KUKA KRL program: kuka-srfPath001.src

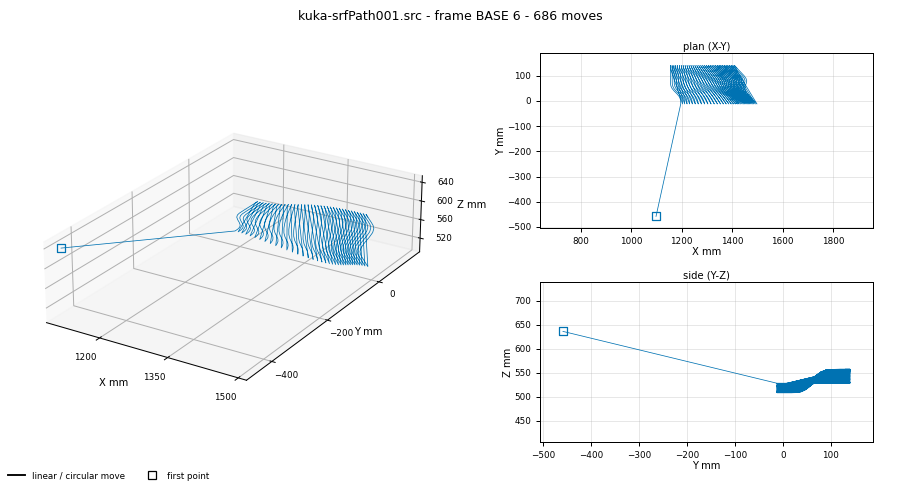
[picture p0: tool path of kuka-srfPath001.src in frame BASE 6, 686 of 688 moves have a stored position in this frame; points joined in program order, loops and branches not executed]
&ACCESS RVP
&REL 1
&PARAM TEMPLATE = C:\KRC\Roboter\Template\vorgabe
&PARAM EDITMASK = *
DEF kuka-srfPath001 ( )
;FOLD INI
;FOLD BASISTECH INI
GLOBAL INTERRUPT DECL 3 WHEN $STOPMESS==TRUE DO IR_STOPM ( )
INTERRUPT ON 3
BAS (#INITMOV,0 )
;ENDFOLD (BASISTECH INI)
;ENDFOLD (INI)
;FOLD STARTPOSITION PTP, VEL 50%, A1 5,A2 -90,A3 100,A4 5,A5 10,A6 -5,E1 0
$BWDSTART = FALSE
PDAT_ACT = {VEL 50,ACC 100,APO_DIST 100}
FDAT_ACT = {TOOL_NO 0,BASE_NO 0,IPO_FRAME #BASE}
BAS (#PTP_PARAMS,50)
$H_POS = {A1 5,A2 -90,A3 100,A4 5,A5 10,A6 -5,E1 0 ,E2 0,E3 0,E4 0,E5 0,E6 0}
PTP  {A1 5,A2 -90,A3 100,A4 5,A5 10,A6 -5,E1 0 ,E2 0,E3 0,E4 0,E5 0,E6 0}
;ENDFOLD
;FOLD SET SPEED TO 50% PTP AND 1 m/sec. LIN
$VEL.CP=1
BAS(#VEL_PTP,50)
BAS(#TOOL,6)
BAS(#BASE,6)
;ENDFOLD
;FOLD PTP FIRST POSITION, VEL= 50 %, TOOL[6], BASE[6]
$BWDSTART = FALSE
PDAT_ACT = {VEL 50,ACC 100,APO_DIST 100}
FDAT_ACT = {TOOL_NO 6,BASE_NO 6,IPO_FRAME #BASE}
BAS (#PTP_PARAMS,50)
;ENDFOLD
PTP {E6POS: X 1098.000, Y -458.000, Z 636.000, A 0.000, B 90.000, C -32.958, E1 0.000, E2 0.0, E3 0.0, E4 0.0, E5 0.0, E6 0.0}
LIN {E6POS: X 1098.000, Y -458.000, Z 636.000, A 0.000, B 90.000, C -32.958, E1 0.000, E2 0.0, E3 0.0, E4 0.0, E5 0.0, E6 0.0} C_DIS
>>>>>>>>>>>>>>>>>>>>>>>>>>>>POWDER FEED ON at=END
>>>>>>>>>>>>>>>>>>>>>>>>>>>>GAS SUPPLY ON at=END
>>>>>>>>>>>>>>>>>>>>>>>>>>>>LASER ON at=END
LIN {E6POS: X 1196.000, Y -12.200, Z 528.000, A 0.000, B 90.000, C -180.000, E1 0.000, E2 0.0, E3 0.0, E4 0.0, E5 0.0, E6 0.0} C_DIS
;POWDER FEED RATE  =  3.0
;LASER INTENSITY  =  4.0
LIN {E6POS: X 1195.747, Y -2.040, Z 528.000, A 90.000, B 90.000, C -90.000, E1 0.000, E2 0.0, E3 0.0, E4 0.0, E5 0.0, E6 0.0} C_DIS
;POWDER FEED RATE  =  3.0
;LASER INTENSITY  =  4.0
LIN {E6POS: X 1193.975, Y 8.120, Z 528.000, A 90.000, B 90.000, C -90.000, E1 0.000, E2 0.0, E3 0.0, E4 0.0, E5 0.0, E6 0.0} C_DIS
;POWDER FEED RATE  =  3.0
;LASER INTENSITY  =  4.0
LIN {E6POS: X 1189.167, Y 18.280, Z 528.000, A -90.000, B 90.000, C 90.000, E1 0.000, E2 0.0, E3 0.0, E4 0.0, E5 0.0, E6 0.0} C_DIS
;POWDER FEED RATE  =  3.0
;LASER INTENSITY  =  4.0
LIN {E6POS: X 1180.562, Y 28.440, Z 528.000, A 90.000, B 90.000, C -90.000, E1 0.000, E2 0.0, E3 0.0, E4 0.0, E5 0.0, E6 0.0} C_DIS
;POWDER FEED RATE  =  3.0
;LASER INTENSITY  =  4.0
LIN {E6POS: X 1170.438, Y 38.600, Z 528.000, A 0.000, B 90.000, C -180.000, E1 0.000, E2 0.0, E3 0.0, E4 0.0, E5 0.0, E6 0.0} C_DIS
;POWDER FEED RATE  =  3.0
;LASER INTENSITY  =  4.0
LIN {E6POS: X 1161.833, Y 48.760, Z 528.000, A 0.000, B 90.000, C -180.000, E1 0.000, E2 0.0, E3 0.0, E4 0.0, E5 0.0, E6 0.0} C_DIS
;POWDER FEED RATE  =  3.0
;LASER INTENSITY  =  4.0
LIN {E6POS: X 1157.025, Y 58.920, Z 528.000, A 0.000, B 90.000, C -180.000, E1 0.000, E2 0.0, E3 0.0, E4 0.0, E5 0.0, E6 0.0} C_DIS
;POWDER FEED RATE  =  3.0
;LASER INTENSITY  =  4.0
LIN {E6POS: X 1155.253, Y 69.080, Z 528.000, A 0.000, B 90.000, C -180.000, E1 0.000, E2 0.0, E3 0.0, E4 0.0, E5 0.0, E6 0.0} C_DIS
;POWDER FEED RATE  =  3.0
;LASER INTENSITY  =  4.0
LIN {E6POS: X 1155.000, Y 79.240, Z 528.000, A 0.000, B 90.000, C -180.000, E1 0.000, E2 0.0, E3 0.0, E4 0.0, E5 0.0, E6 0.0} C_DIS
;POWDER FEED RATE  =  3.0
;LASER INTENSITY  =  4.0
LIN {E6POS: X 1155.000, Y 89.400, Z 528.000, A 0.000, B 90.000, C -180.000, E1 0.000, E2 0.0, E3 0.0, E4 0.0, E5 0.0, E6 0.0} C_DIS
;POWDER FEED RATE  =  3.0
;LASER INTENSITY  =  4.0
LIN {E6POS: X 1155.000, Y 99.560, Z 528.000, A 0.000, B 90.000, C -180.000, E1 0.000, E2 0.0, E3 0.0, E4 0.0, E5 0.0, E6 0.0} C_DIS
;POWDER FEED RATE  =  3.0
;LASER INTENSITY  =  4.0
LIN {E6POS: X 1155.000, Y 109.720, Z 528.000, A 0.000, B 90.000, C -180.000, E1 0.000, E2 0.0, E3 0.0, E4 0.0, E5 0.0, E6 0.0} C_DIS
;POWDER FEED RATE  =  3.0
;LASER INTENSITY  =  4.0
LIN {E6POS: X 1155.000, Y 119.880, Z 528.000, A 0.000, B 90.000, C -180.000, E1 0.000, E2 0.0, E3 0.0, E4 0.0, E5 0.0, E6 0.0} C_DIS
;POWDER FEED RATE  =  3.0
;LASER INTENSITY  =  4.0
LIN {E6POS: X 1155.000, Y 130.040, Z 528.000, A 0.000, B 90.000, C -180.000, E1 0.000, E2 0.0, E3 0.0, E4 0.0, E5 0.0, E6 0.0} C_DIS
;POWDER FEED RATE  =  3.0
;LASER INTENSITY  =  4.0
LIN {E6POS: X 1155.000, Y 140.200, Z 528.000, A 0.000, B 90.000, C -180.000, E1 0.000, E2 0.0, E3 0.0, E4 0.0, E5 0.0, E6 0.0} C_DIS
;POWDER FEED RATE  =  3.0
;LASER INTENSITY  =  4.0
>>>>>>>>>>>>>>>>>>>>>>>>>>>>POWDER FEED OFF  at=START
>>>>>>>>>>>>>>>>>>>>>>>>>>>>LASER OFF at=START
>>>>>>>>>>>>>>>>>>>>>>>>>>>>GAS SUPPLY OFF  at=START
LIN {E6POS: X 1155.000, Y 140.200, Z 528.000, A 0.000, B 90.000, C -180.000, E1 0.000, E2 0.0, E3 0.0, E4 0.0, E5 0.0, E6 0.0} C_DIS
LIN {E6POS: X 1155.000, Y 130.040, Z 528.000, A 0.000, B 90.000, C -180.000, E1 0.000, E2 0.0, E3 0.0, E4 0.0, E5 0.0, E6 0.0} C_DIS
LIN {E6POS: X 1155.000, Y 130.040, Z 528.000, A 0.000, B 90.000, C -180.000, E1 0.000, E2 0.0, E3 0.0, E4 0.0, E5 0.0, E6 0.0} C_DIS
>>>>>>>>>>>>>>>>>>>>>>>>>>>>GAS SUPPLY ON at=END
>>>>>>>>>>>>>>>>>>>>>>>>>>>>POWDER FEED ON at=END
>>>>>>>>>>>>>>>>>>>>>>>>>>>>LASER ON at=END
LIN {E6POS: X 1203.323, Y -12.200, Z 527.825, A -179.740, B 87.512, C 0.260, E1 0.000, E2 0.0, E3 0.0, E4 0.0, E5 0.0, E6 0.0} C_DIS
;POWDER FEED RATE  =  3.0
;LASER INTENSITY  =  4.0
LIN {E6POS: X 1203.025, Y -2.040, Z 527.825, A -175.488, B 87.476, C 4.508, E1 0.000, E2 0.0, E3 0.0, E4 0.0, E5 0.0, E6 0.0} C_DIS
;POWDER FEED RATE  =  3.0
;LASER INTENSITY  =  4.0
LIN {E6POS: X 1201.215, Y 8.120, Z 527.825, A -163.194, B 87.347, C 16.789, E1 0.000, E2 0.0, E3 0.0, E4 0.0, E5 0.0, E6 0.0} C_DIS
;POWDER FEED RATE  =  3.0
;LASER INTENSITY  =  4.0
LIN {E6POS: X 1196.383, Y 18.280, Z 527.825, A -146.024, B 86.920, C 33.938, E1 0.000, E2 0.0, E3 0.0, E4 0.0, E5 0.0, E6 0.0} C_DIS
;POWDER FEED RATE  =  3.0
;LASER INTENSITY  =  4.0
LIN {E6POS: X 1187.773, Y 28.440, Z 527.827, A -136.214, B 86.497, C 43.733, E1 0.000, E2 0.0, E3 0.0, E4 0.0, E5 0.0, E6 0.0} C_DIS
;POWDER FEED RATE  =  3.0
;LASER INTENSITY  =  4.0
LIN {E6POS: X 1177.652, Y 38.600, Z 527.841, A -137.529, B 86.842, C 42.428, E1 0.000, E2 0.0, E3 0.0, E4 0.0, E5 0.0, E6 0.0} C_DIS
;POWDER FEED RATE  =  3.0
;LASER INTENSITY  =  4.0
LIN {E6POS: X 1169.042, Y 48.760, Z 527.878, A -152.965, B 87.985, C 27.020, E1 0.000, E2 0.0, E3 0.0, E4 0.0, E5 0.0, E6 0.0} C_DIS
;POWDER FEED RATE  =  3.0
;LASER INTENSITY  =  4.0
LIN {E6POS: X 1164.211, Y 58.920, Z 527.943, A 168.385, B 89.147, C -11.614, E1 0.000, E2 0.0, E3 0.0, E4 0.0, E5 0.0, E6 0.0} C_DIS
;POWDER FEED RATE  =  3.0
;LASER INTENSITY  =  4.0
LIN {E6POS: X 1162.402, Y 69.080, Z 528.020, A 55.505, B 89.456, C -124.496, E1 0.000, E2 0.0, E3 0.0, E4 0.0, E5 0.0, E6 0.0} C_DIS
;POWDER FEED RATE  =  3.0
;LASER INTENSITY  =  4.0
LIN {E6POS: X 1162.105, Y 79.240, Z 528.086, A 12.952, B 88.664, C -167.052, E1 0.000, E2 0.0, E3 0.0, E4 0.0, E5 0.0, E6 0.0} C_DIS
;POWDER FEED RATE  =  3.0
;LASER INTENSITY  =  4.0
LIN {E6POS: X 1162.059, Y 89.400, Z 528.123, A 4.232, B 88.116, C -175.770, E1 0.000, E2 0.0, E3 0.0, E4 0.0, E5 0.0, E6 0.0} C_DIS
;POWDER FEED RATE  =  3.0
;LASER INTENSITY  =  4.0
LIN {E6POS: X 1162.013, Y 99.560, Z 528.136, A 1.145, B 87.889, C -178.856, E1 0.000, E2 0.0, E3 0.0, E4 0.0, E5 0.0, E6 0.0} C_DIS
;POWDER FEED RATE  =  3.0
;LASER INTENSITY  =  4.0
LIN {E6POS: X 1161.967, Y 109.720, Z 528.138, A 0.260, B 87.832, C -179.740, E1 0.000, E2 0.0, E3 0.0, E4 0.0, E5 0.0, E6 0.0} C_DIS
;POWDER FEED RATE  =  3.0
;LASER INTENSITY  =  4.0
LIN {E6POS: X 1161.921, Y 119.880, Z 528.138, A 0.260, B 87.805, C -179.740, E1 0.000, E2 0.0, E3 0.0, E4 0.0, E5 0.0, E6 0.0} C_DIS
;POWDER FEED RATE  =  3.0
;LASER INTENSITY  =  4.0
LIN {E6POS: X 1161.875, Y 130.040, Z 528.138, A 0.260, B 87.776, C -179.740, E1 0.000, E2 0.0, E3 0.0, E4 0.0, E5 0.0, E6 0.0} C_DIS
;POWDER FEED RATE  =  3.0
;LASER INTENSITY  =  4.0
LIN {E6POS: X 1161.829, Y 140.200, Z 528.138, A 0.260, B 87.747, C -179.740, E1 0.000, E2 0.0, E3 0.0, E4 0.0, E5 0.0, E6 0.0} C_DIS
;POWDER FEED RATE  =  3.0
;LASER INTENSITY  =  4.0
>>>>>>>>>>>>>>>>>>>>>>>>>>>>POWDER FEED OFF  at=START
>>>>>>>>>>>>>>>>>>>>>>>>>>>>LASER OFF at=START
>>>>>>>>>>>>>>>>>>>>>>>>>>>>GAS SUPPLY OFF  at=START
LIN {E6POS: X 1161.829, Y 140.200, Z 528.138, A 0.260, B 87.747, C -179.740, E1 0.000, E2 0.0, E3 0.0, E4 0.0, E5 0.0, E6 0.0} C_DIS
LIN {E6POS: X 1161.875, Y 130.040, Z 528.138, A 0.260, B 87.776, C -179.740, E1 0.000, E2 0.0, E3 0.0, E4 0.0, E5 0.0, E6 0.0} C_DIS
LIN {E6POS: X 1161.875, Y 130.040, Z 528.138, A 0.260, B 87.776, C -179.740, E1 0.000, E2 0.0, E3 0.0, E4 0.0, E5 0.0, E6 0.0} C_DIS
>>>>>>>>>>>>>>>>>>>>>>>>>>>>GAS SUPPLY ON at=END
>>>>>>>>>>>>>>>>>>>>>>>>>>>>POWDER FEED ON at=END
>>>>>>>>>>>>>>>>>>>>>>>>>>>>LASER ON at=END
LIN {E6POS: X 1211.725, Y -12.200, Z 527.328, A -178.991, B 85.857, C 1.007, E1 0.000, E2 0.0, E3 0.0, E4 0.0, E5 0.0, E6 0.0} C_DIS
;POWDER FEED RATE  =  3.0
;LASER INTENSITY  =  4.0
LIN {E6POS: X 1211.298, Y -2.040, Z 527.328, A -174.802, B 85.760, C 5.184, E1 0.000, E2 0.0, E3 0.0, E4 0.0, E5 0.0, E6 0.0} C_DIS
;POWDER FEED RATE  =  3.0
;LASER INTENSITY  =  4.0
LIN {E6POS: X 1209.380, Y 8.120, Z 527.328, A -162.723, B 85.506, C 17.227, E1 0.000, E2 0.0, E3 0.0, E4 0.0, E5 0.0, E6 0.0} C_DIS
;POWDER FEED RATE  =  3.0
;LASER INTENSITY  =  4.0
LIN {E6POS: X 1204.481, Y 18.280, Z 527.328, A -145.872, B 84.767, C 34.017, E1 0.000, E2 0.0, E3 0.0, E4 0.0, E5 0.0, E6 0.0} C_DIS
;POWDER FEED RATE  =  3.0
;LASER INTENSITY  =  4.0
LIN {E6POS: X 1195.856, Y 28.440, Z 527.336, A -136.715, B 84.106, C 43.133, E1 0.000, E2 0.0, E3 0.0, E4 0.0, E5 0.0, E6 0.0} C_DIS
;POWDER FEED RATE  =  3.0
;LASER INTENSITY  =  4.0
LIN {E6POS: X 1185.742, Y 38.600, Z 527.388, A -139.845, B 84.831, C 40.040, E1 0.000, E2 0.0, E3 0.0, E4 0.0, E5 0.0, E6 0.0} C_DIS
;POWDER FEED RATE  =  3.0
;LASER INTENSITY  =  4.0
LIN {E6POS: X 1177.119, Y 48.760, Z 527.530, A -163.042, B 86.819, C 16.934, E1 0.000, E2 0.0, E3 0.0, E4 0.0, E5 0.0, E6 0.0} C_DIS
;POWDER FEED RATE  =  3.0
;LASER INTENSITY  =  4.0
LIN {E6POS: X 1172.225, Y 58.920, Z 527.783, A 139.529, B 88.149, C -40.456, E1 0.000, E2 0.0, E3 0.0, E4 0.0, E5 0.0, E6 0.0} C_DIS
;POWDER FEED RATE  =  3.0
;LASER INTENSITY  =  4.0
LIN {E6POS: X 1170.312, Y 69.080, Z 528.081, A 71.606, B 88.220, C -108.402, E1 0.000, E2 0.0, E3 0.0, E4 0.0, E5 0.0, E6 0.0} C_DIS
;POWDER FEED RATE  =  3.0
;LASER INTENSITY  =  4.0
LIN {E6POS: X 1169.889, Y 79.240, Z 528.334, A 27.036, B 87.418, C -152.987, E1 0.000, E2 0.0, E3 0.0, E4 0.0, E5 0.0, E6 0.0} C_DIS
;POWDER FEED RATE  =  3.0
;LASER INTENSITY  =  4.0
LIN {E6POS: X 1169.712, Y 89.400, Z 528.476, A 9.569, B 86.620, C -170.447, E1 0.000, E2 0.0, E3 0.0, E4 0.0, E5 0.0, E6 0.0} C_DIS
;POWDER FEED RATE  =  3.0
;LASER INTENSITY  =  4.0
LIN {E6POS: X 1169.534, Y 99.560, Z 528.528, A 2.915, B 86.218, C -177.092, E1 0.000, E2 0.0, E3 0.0, E4 0.0, E5 0.0, E6 0.0} C_DIS
;POWDER FEED RATE  =  3.0
;LASER INTENSITY  =  4.0
LIN {E6POS: X 1169.355, Y 109.720, Z 528.536, A 1.009, B 86.082, C -178.993, E1 0.000, E2 0.0, E3 0.0, E4 0.0, E5 0.0, E6 0.0} C_DIS
;POWDER FEED RATE  =  3.0
;LASER INTENSITY  =  4.0
LIN {E6POS: X 1169.176, Y 119.880, Z 528.536, A 1.009, B 85.991, C -178.993, E1 0.000, E2 0.0, E3 0.0, E4 0.0, E5 0.0, E6 0.0} C_DIS
;POWDER FEED RATE  =  3.0
;LASER INTENSITY  =  4.0
LIN {E6POS: X 1168.997, Y 130.040, Z 528.536, A 1.009, B 85.895, C -178.993, E1 0.000, E2 0.0, E3 0.0, E4 0.0, E5 0.0, E6 0.0} C_DIS
;POWDER FEED RATE  =  3.0
;LASER INTENSITY  =  4.0
LIN {E6POS: X 1168.818, Y 140.200, Z 528.536, A 1.009, B 85.794, C -178.993, E1 0.000, E2 0.0, E3 0.0, E4 0.0, E5 0.0, E6 0.0} C_DIS
;POWDER FEED RATE  =  3.0
;LASER INTENSITY  =  4.0
>>>>>>>>>>>>>>>>>>>>>>>>>>>>POWDER FEED OFF  at=START
>>>>>>>>>>>>>>>>>>>>>>>>>>>>LASER OFF at=START
>>>>>>>>>>>>>>>>>>>>>>>>>>>>GAS SUPPLY OFF  at=START
LIN {E6POS: X 1168.818, Y 140.200, Z 528.536, A 1.009, B 85.794, C -178.993, E1 0.000, E2 0.0, E3 0.0, E4 0.0, E5 0.0, E6 0.0} C_DIS
LIN {E6POS: X 1168.997, Y 130.040, Z 528.536, A 1.009, B 85.895, C -178.993, E1 0.000, E2 0.0, E3 0.0, E4 0.0, E5 0.0, E6 0.0} C_DIS
LIN {E6POS: X 1168.997, Y 130.040, Z 528.536, A 1.009, B 85.895, C -178.993, E1 0.000, E2 0.0, E3 0.0, E4 0.0, E5 0.0, E6 0.0} C_DIS
>>>>>>>>>>>>>>>>>>>>>>>>>>>>GAS SUPPLY ON at=END
>>>>>>>>>>>>>>>>>>>>>>>>>>>>POWDER FEED ON at=END
>>>>>>>>>>>>>>>>>>>>>>>>>>>>LASER ON at=END
LIN {E6POS: X 1221.090, Y -12.200, Z 526.549, A -177.798, B 84.710, C 2.192, E1 0.000, E2 0.0, E3 0.0, E4 0.0, E5 0.0, E6 0.0} C_DIS
;POWDER FEED RATE  =  3.0
;LASER INTENSITY  =  4.0
LIN {E6POS: X 1220.457, Y -2.040, Z 526.549, A -173.713, B 84.549, C 6.258, E1 0.000, E2 0.0, E3 0.0, E4 0.0, E5 0.0, E6 0.0} C_DIS
;POWDER FEED RATE  =  3.0
;LASER INTENSITY  =  4.0
LIN {E6POS: X 1218.366, Y 8.120, Z 526.549, A -161.979, B 84.181, C 17.934, E1 0.000, E2 0.0, E3 0.0, E4 0.0, E5 0.0, E6 0.0} C_DIS
;POWDER FEED RATE  =  3.0
;LASER INTENSITY  =  4.0
LIN {E6POS: X 1213.360, Y 18.280, Z 526.549, A -145.631, B 83.214, C 34.181, E1 0.000, E2 0.0, E3 0.0, E4 0.0, E5 0.0, E6 0.0} C_DIS
;POWDER FEED RATE  =  3.0
;LASER INTENSITY  =  4.0
LIN {E6POS: X 1204.712, Y 28.440, Z 526.565, A -137.335, B 82.454, C 42.417, E1 0.000, E2 0.0, E3 0.0, E4 0.0, E5 0.0, E6 0.0} C_DIS
;POWDER FEED RATE  =  3.0
;LASER INTENSITY  =  4.0
LIN {E6POS: X 1194.609, Y 38.600, Z 526.678, A -142.877, B 83.593, C 36.951, E1 0.000, E2 0.0, E3 0.0, E4 0.0, E5 0.0, E6 0.0} C_DIS
;POWDER FEED RATE  =  3.0
;LASER INTENSITY  =  4.0
LIN {E6POS: X 1185.969, Y 48.760, Z 526.986, A -176.728, B 86.064, C 3.265, E1 0.000, E2 0.0, E3 0.0, E4 0.0, E5 0.0, E6 0.0} C_DIS
;POWDER FEED RATE  =  3.0
;LASER INTENSITY  =  4.0
LIN {E6POS: X 1180.978, Y 58.920, Z 527.536, A 121.216, B 86.528, C -58.738, E1 0.000, E2 0.0, E3 0.0, E4 0.0, E5 0.0, E6 0.0} C_DIS
;POWDER FEED RATE  =  3.0
;LASER INTENSITY  =  4.0
LIN {E6POS: X 1178.905, Y 69.080, Z 528.182, A 77.896, B 86.281, C -102.128, E1 0.000, E2 0.0, E3 0.0, E4 0.0, E5 0.0, E6 0.0} C_DIS
;POWDER FEED RATE  =  3.0
;LASER INTENSITY  =  4.0
LIN {E6POS: X 1178.286, Y 79.240, Z 528.732, A 39.861, B 85.985, C -140.208, E1 0.000, E2 0.0, E3 0.0, E4 0.0, E5 0.0, E6 0.0} C_DIS
;POWDER FEED RATE  =  3.0
;LASER INTENSITY  =  4.0
LIN {E6POS: X 1177.904, Y 89.400, Z 529.039, A 15.736, B 85.348, C -164.313, E1 0.000, E2 0.0, E3 0.0, E4 0.0, E5 0.0, E6 0.0} C_DIS
;POWDER FEED RATE  =  3.0
;LASER INTENSITY  =  4.0
LIN {E6POS: X 1177.516, Y 99.560, Z 529.153, A 5.242, B 84.872, C -174.779, E1 0.000, E2 0.0, E3 0.0, E4 0.0, E5 0.0, E6 0.0} C_DIS
;POWDER FEED RATE  =  3.0
;LASER INTENSITY  =  4.0
LIN {E6POS: X 1177.126, Y 109.720, Z 529.169, A 2.202, B 84.658, C -177.808, E1 0.000, E2 0.0, E3 0.0, E4 0.0, E5 0.0, E6 0.0} C_DIS
;POWDER FEED RATE  =  3.0
;LASER INTENSITY  =  4.0
LIN {E6POS: X 1176.735, Y 119.880, Z 529.169, A 2.202, B 84.487, C -177.808, E1 0.000, E2 0.0, E3 0.0, E4 0.0, E5 0.0, E6 0.0} C_DIS
;POWDER FEED RATE  =  3.0
;LASER INTENSITY  =  4.0
LIN {E6POS: X 1176.345, Y 130.040, Z 529.169, A 2.202, B 84.305, C -177.809, E1 0.000, E2 0.0, E3 0.0, E4 0.0, E5 0.0, E6 0.0} C_DIS
;POWDER FEED RATE  =  3.0
;LASER INTENSITY  =  4.0
LIN {E6POS: X 1175.954, Y 140.200, Z 529.169, A 2.202, B 84.110, C -177.810, E1 0.000, E2 0.0, E3 0.0, E4 0.0, E5 0.0, E6 0.0} C_DIS
;POWDER FEED RATE  =  3.0
;LASER INTENSITY  =  4.0
>>>>>>>>>>>>>>>>>>>>>>>>>>>>POWDER FEED OFF  at=START
>>>>>>>>>>>>>>>>>>>>>>>>>>>>LASER OFF at=START
>>>>>>>>>>>>>>>>>>>>>>>>>>>>GAS SUPPLY OFF  at=START
LIN {E6POS: X 1175.954, Y 140.200, Z 529.169, A 2.202, B 84.110, C -177.810, E1 0.000, E2 0.0, E3 0.0, E4 0.0, E5 0.0, E6 0.0} C_DIS
LIN {E6POS: X 1176.345, Y 130.040, Z 529.169, A 2.202, B 84.305, C -177.809, E1 0.000, E2 0.0, E3 0.0, E4 0.0, E5 0.0, E6 0.0} C_DIS
LIN {E6POS: X 1176.345, Y 130.040, Z 529.169, A 2.202, B 84.305, C -177.809, E1 0.000, E2 0.0, E3 0.0, E4 0.0, E5 0.0, E6 0.0} C_DIS
>>>>>>>>>>>>>>>>>>>>>>>>>>>>GAS SUPPLY ON at=END
>>>>>>>>>>>>>>>>>>>>>>>>>>>>POWDER FEED ON at=END
>>>>>>>>>>>>>>>>>>>>>>>>>>>>LASER ON at=END
LIN {E6POS: X 1231.298, Y -12.200, Z 525.527, A -176.212, B 83.899, C 3.767, E1 0.000, E2 0.0, E3 0.0, E4 0.0, E5 0.0, E6 0.0} C_DIS
;POWDER FEED RATE  =  3.0
;LASER INTENSITY  =  4.0
LIN {E6POS: X 1230.390, Y -2.040, Z 525.527, A -172.269, B 83.675, C 7.684, E1 0.000, E2 0.0, E3 0.0, E4 0.0, E5 0.0, E6 0.0} C_DIS
;POWDER FEED RATE  =  3.0
;LASER INTENSITY  =  4.0
LIN {E6POS: X 1228.069, Y 8.120, Z 525.527, A -160.997, B 83.205, C 18.879, E1 0.000, E2 0.0, E3 0.0, E4 0.0, E5 0.0, E6 0.0} C_DIS
;POWDER FEED RATE  =  3.0
;LASER INTENSITY  =  4.0
LIN {E6POS: X 1222.921, Y 18.280, Z 525.527, A -145.313, B 82.075, C 34.430, E1 0.000, E2 0.0, E3 0.0, E4 0.0, E5 0.0, E6 0.0} C_DIS
;POWDER FEED RATE  =  3.0
;LASER INTENSITY  =  4.0
LIN {E6POS: X 1214.242, Y 28.440, Z 525.555, A -138.077, B 81.322, C 41.595, E1 0.000, E2 0.0, E3 0.0, E4 0.0, E5 0.0, E6 0.0} C_DIS
;POWDER FEED RATE  =  3.0
;LASER INTENSITY  =  4.0
LIN {E6POS: X 1204.156, Y 38.600, Z 525.749, A -146.760, B 82.894, C 33.038, E1 0.000, E2 0.0, E3 0.0, E4 0.0, E5 0.0, E6 0.0} C_DIS
;POWDER FEED RATE  =  3.0
;LASER INTENSITY  =  4.0
LIN {E6POS: X 1195.495, Y 48.760, Z 526.275, A 166.884, B 85.317, C -13.074, E1 0.000, E2 0.0, E3 0.0, E4 0.0, E5 0.0, E6 0.0} C_DIS
;POWDER FEED RATE  =  3.0
;LASER INTENSITY  =  4.0
LIN {E6POS: X 1190.382, Y 58.920, Z 527.216, A 110.981, B 84.250, C -68.922, E1 0.000, E2 0.0, E3 0.0, E4 0.0, E5 0.0, E6 0.0} C_DIS
;POWDER FEED RATE  =  3.0
;LASER INTENSITY  =  4.0
LIN {E6POS: X 1188.102, Y 69.080, Z 528.324, A 81.066, B 83.730, C -98.987, E1 0.000, E2 0.0, E3 0.0, E4 0.0, E5 0.0, E6 0.0} C_DIS
;POWDER FEED RATE  =  3.0
;LASER INTENSITY  =  4.0
LIN {E6POS: X 1187.229, Y 79.240, Z 529.265, A 50.146, B 84.221, C -129.997, E1 0.000, E2 0.0, E3 0.0, E4 0.0, E5 0.0, E6 0.0} C_DIS
;POWDER FEED RATE  =  3.0
;LASER INTENSITY  =  4.0
LIN {E6POS: X 1186.576, Y 89.400, Z 529.791, A 22.371, B 84.174, C -157.733, E1 0.000, E2 0.0, E3 0.0, E4 0.0, E5 0.0, E6 0.0} C_DIS
;POWDER FEED RATE  =  3.0
;LASER INTENSITY  =  4.0
LIN {E6POS: X 1185.911, Y 99.560, Z 529.985, A 8.053, B 83.765, C -171.994, E1 0.000, E2 0.0, E3 0.0, E4 0.0, E5 0.0, E6 0.0} C_DIS
;POWDER FEED RATE  =  3.0
;LASER INTENSITY  =  4.0
LIN {E6POS: X 1185.239, Y 109.720, Z 530.013, A 3.788, B 83.492, C -176.236, E1 0.000, E2 0.0, E3 0.0, E4 0.0, E5 0.0, E6 0.0} C_DIS
;POWDER FEED RATE  =  3.0
;LASER INTENSITY  =  4.0
LIN {E6POS: X 1184.566, Y 119.880, Z 530.013, A 3.788, B 83.237, C -176.238, E1 0.000, E2 0.0, E3 0.0, E4 0.0, E5 0.0, E6 0.0} C_DIS
;POWDER FEED RATE  =  3.0
;LASER INTENSITY  =  4.0
LIN {E6POS: X 1183.894, Y 130.040, Z 530.013, A 3.788, B 82.961, C -176.240, E1 0.000, E2 0.0, E3 0.0, E4 0.0, E5 0.0, E6 0.0} C_DIS
;POWDER FEED RATE  =  3.0
;LASER INTENSITY  =  4.0
LIN {E6POS: X 1183.221, Y 140.200, Z 530.013, A 3.788, B 82.662, C -176.243, E1 0.000, E2 0.0, E3 0.0, E4 0.0, E5 0.0, E6 0.0} C_DIS
;POWDER FEED RATE  =  3.0
;LASER INTENSITY  =  4.0
>>>>>>>>>>>>>>>>>>>>>>>>>>>>POWDER FEED OFF  at=START
>>>>>>>>>>>>>>>>>>>>>>>>>>>>LASER OFF at=START
>>>>>>>>>>>>>>>>>>>>>>>>>>>>GAS SUPPLY OFF  at=START
LIN {E6POS: X 1183.221, Y 140.200, Z 530.013, A 3.788, B 82.662, C -176.243, E1 0.000, E2 0.0, E3 0.0, E4 0.0, E5 0.0, E6 0.0} C_DIS
LIN {E6POS: X 1183.894, Y 130.040, Z 530.013, A 3.788, B 82.961, C -176.240, E1 0.000, E2 0.0, E3 0.0, E4 0.0, E5 0.0, E6 0.0} C_DIS
LIN {E6POS: X 1183.894, Y 130.040, Z 530.013, A 3.788, B 82.961, C -176.240, E1 0.000, E2 0.0, E3 0.0, E4 0.0, E5 0.0, E6 0.0} C_DIS
>>>>>>>>>>>>>>>>>>>>>>>>>>>>GAS SUPPLY ON at=END
>>>>>>>>>>>>>>>>>>>>>>>>>>>>POWDER FEED ON at=END
>>>>>>>>>>>>>>>>>>>>>>>>>>>>LASER ON at=END
LIN {E6POS: X 1242.232, Y -12.200, Z 524.303, A -174.283, B 83.319, C 5.679, E1 0.000, E2 0.0, E3 0.0, E4 0.0, E5 0.0, E6 0.0} C_DIS
;POWDER FEED RATE  =  3.0
;LASER INTENSITY  =  4.0
LIN {E6POS: X 1240.988, Y -2.040, Z 524.303, A -170.519, B 83.038, C 9.413, E1 0.000, E2 0.0, E3 0.0, E4 0.0, E5 0.0, E6 0.0} C_DIS
;POWDER FEED RATE  =  3.0
;LASER INTENSITY  =  4.0
LIN {E6POS: X 1238.385, Y 8.120, Z 524.303, A -159.813, B 82.480, C 20.027, E1 0.000, E2 0.0, E3 0.0, E4 0.0, E5 0.0, E6 0.0} C_DIS
;POWDER FEED RATE  =  3.0
;LASER INTENSITY  =  4.0
LIN {E6POS: X 1233.064, Y 18.280, Z 524.303, A -144.927, B 81.238, C 34.757, E1 0.000, E2 0.0, E3 0.0, E4 0.0, E5 0.0, E6 0.0} C_DIS
;POWDER FEED RATE  =  3.0
;LASER INTENSITY  =  4.0
LIN {E6POS: X 1224.347, Y 28.440, Z 524.345, A -138.947, B 80.574, C 40.668, E1 0.000, E2 0.0, E3 0.0, E4 0.0, E5 0.0, E6 0.0} C_DIS
;POWDER FEED RATE  =  3.0
;LASER INTENSITY  =  4.0
LIN {E6POS: X 1214.283, Y 38.600, Z 524.636, A -151.669, B 82.570, C 28.129, E1 0.000, E2 0.0, E3 0.0, E4 0.0, E5 0.0, E6 0.0} C_DIS
;POWDER FEED RATE  =  3.0
;LASER INTENSITY  =  4.0
LIN {E6POS: X 1205.602, Y 48.760, Z 525.427, A 150.464, B 84.256, C -29.412, E1 0.000, E2 0.0, E3 0.0, E4 0.0, E5 0.0, E6 0.0} C_DIS
;POWDER FEED RATE  =  3.0
;LASER INTENSITY  =  4.0
LIN {E6POS: X 1200.350, Y 58.920, Z 526.841, A 104.954, B 81.423, C -74.884, E1 0.000, E2 0.0, E3 0.0, E4 0.0, E5 0.0, E6 0.0} C_DIS
;POWDER FEED RATE  =  3.0
;LASER INTENSITY  =  4.0
LIN {E6POS: X 1197.827, Y 69.080, Z 528.506, A 82.914, B 80.675, C -97.180, E1 0.000, E2 0.0, E3 0.0, E4 0.0, E5 0.0, E6 0.0} C_DIS
;POWDER FEED RATE  =  3.0
;LASER INTENSITY  =  4.0
LIN {E6POS: X 1196.652, Y 79.240, Z 529.920, A 57.886, B 82.098, C -122.360, E1 0.000, E2 0.0, E3 0.0, E4 0.0, E5 0.0, E6 0.0} C_DIS
;POWDER FEED RATE  =  3.0
;LASER INTENSITY  =  4.0
LIN {E6POS: X 1195.673, Y 89.400, Z 530.711, A 29.078, B 83.006, C -151.103, E1 0.000, E2 0.0, E3 0.0, E4 0.0, E5 0.0, E6 0.0} C_DIS
;POWDER FEED RATE  =  3.0
;LASER INTENSITY  =  4.0
LIN {E6POS: X 1194.670, Y 99.560, Z 531.002, A 11.262, B 82.831, C -168.824, E1 0.000, E2 0.0, E3 0.0, E4 0.0, E5 0.0, E6 0.0} C_DIS
;POWDER FEED RATE  =  3.0
;LASER INTENSITY  =  4.0
LIN {E6POS: X 1193.655, Y 109.720, Z 531.044, A 5.717, B 82.530, C -174.331, E1 0.000, E2 0.0, E3 0.0, E4 0.0, E5 0.0, E6 0.0} C_DIS
;POWDER FEED RATE  =  3.0
;LASER INTENSITY  =  4.0
LIN {E6POS: X 1192.638, Y 119.880, Z 531.044, A 5.717, B 82.194, C -174.335, E1 0.000, E2 0.0, E3 0.0, E4 0.0, E5 0.0, E6 0.0} C_DIS
;POWDER FEED RATE  =  3.0
;LASER INTENSITY  =  4.0
LIN {E6POS: X 1191.621, Y 130.040, Z 531.044, A 5.717, B 81.826, C -174.340, E1 0.000, E2 0.0, E3 0.0, E4 0.0, E5 0.0, E6 0.0} C_DIS
;POWDER FEED RATE  =  3.0
;LASER INTENSITY  =  4.0
LIN {E6POS: X 1190.603, Y 140.200, Z 531.044, A 5.717, B 81.422, C -174.346, E1 0.000, E2 0.0, E3 0.0, E4 0.0, E5 0.0, E6 0.0} C_DIS
;POWDER FEED RATE  =  3.0
;LASER INTENSITY  =  4.0
>>>>>>>>>>>>>>>>>>>>>>>>>>>>POWDER FEED OFF  at=START
>>>>>>>>>>>>>>>>>>>>>>>>>>>>LASER OFF at=START
>>>>>>>>>>>>>>>>>>>>>>>>>>>>GAS SUPPLY OFF  at=START
LIN {E6POS: X 1190.603, Y 140.200, Z 531.044, A 5.717, B 81.422, C -174.346, E1 0.000, E2 0.0, E3 0.0, E4 0.0, E5 0.0, E6 0.0} C_DIS
LIN {E6POS: X 1191.621, Y 130.040, Z 531.044, A 5.717, B 81.826, C -174.340, E1 0.000, E2 0.0, E3 0.0, E4 0.0, E5 0.0, E6 0.0} C_DIS
LIN {E6POS: X 1191.621, Y 130.040, Z 531.044, A 5.717, B 81.826, C -174.340, E1 0.000, E2 0.0, E3 0.0, E4 0.0, E5 0.0, E6 0.0} C_DIS
>>>>>>>>>>>>>>>>>>>>>>>>>>>>GAS SUPPLY ON at=END
>>>>>>>>>>>>>>>>>>>>>>>>>>>>POWDER FEED ON at=END
>>>>>>>>>>>>>>>>>>>>>>>>>>>>LASER ON at=END
LIN {E6POS: X 1253.772, Y -12.200, Z 522.917, A -172.066, B 82.909, C 7.874, E1 0.000, E2 0.0, E3 0.0, E4 0.0, E5 0.0, E6 0.0} C_DIS
;POWDER FEED RATE  =  3.0
;LASER INTENSITY  =  4.0
LIN {E6POS: X 1252.140, Y -2.040, Z 522.917, A -168.515, B 82.578, C 11.391, E1 0.000, E2 0.0, E3 0.0, E4 0.0, E5 0.0, E6 0.0} C_DIS
;POWDER FEED RATE  =  3.0
;LASER INTENSITY  =  4.0
LIN {E6POS: X 1249.211, Y 8.120, Z 522.917, A -158.465, B 81.944, C 21.342, E1 0.000, E2 0.0, E3 0.0, E4 0.0, E5 0.0, E6 0.0} C_DIS
;POWDER FEED RATE  =  3.0
;LASER INTENSITY  =  4.0
LIN {E6POS: X 1243.689, Y 18.280, Z 522.917, A -144.486, B 80.635, C 35.152, E1 0.000, E2 0.0, E3 0.0, E4 0.0, E5 0.0, E6 0.0} C_DIS
;POWDER FEED RATE  =  3.0
;LASER INTENSITY  =  4.0
LIN {E6POS: X 1234.929, Y 28.440, Z 522.974, A -139.956, B 80.125, C 39.624, E1 0.000, E2 0.0, E3 0.0, E4 0.0, E5 0.0, E6 0.0} C_DIS
;POWDER FEED RATE  =  3.0
;LASER INTENSITY  =  4.0
LIN {E6POS: X 1224.893, Y 38.600, Z 523.377, A -157.810, B 82.493, C 22.018, E1 0.000, E2 0.0, E3 0.0, E4 0.0, E5 0.0, E6 0.0} C_DIS
;POWDER FEED RATE  =  3.0
;LASER INTENSITY  =  4.0
LIN {E6POS: X 1216.195, Y 48.760, Z 524.470, A 136.592, B 82.733, C -43.178, E1 0.000, E2 0.0, E3 0.0, E4 0.0, E5 0.0, E6 0.0} C_DIS
;POWDER FEED RATE  =  3.0
;LASER INTENSITY  =  4.0
LIN {E6POS: X 1210.792, Y 58.920, Z 526.426, A 101.116, B 78.174, C -78.649, E1 0.000, E2 0.0, E3 0.0, E4 0.0, E5 0.0, E6 0.0} C_DIS
;POWDER FEED RATE  =  3.0
;LASER INTENSITY  =  4.0
LIN {E6POS: X 1208.002, Y 69.080, Z 528.727, A 84.092, B 77.240, C -96.057, E1 0.000, E2 0.0, E3 0.0, E4 0.0, E5 0.0, E6 0.0} C_DIS
;POWDER FEED RATE  =  3.0
;LASER INTENSITY  =  4.0
LIN {E6POS: X 1206.489, Y 79.240, Z 530.684, A 63.606, B 79.659, C -116.769, E1 0.000, E2 0.0, E3 0.0, E4 0.0, E5 0.0, E6 0.0} C_DIS
;POWDER FEED RATE  =  3.0
;LASER INTENSITY  =  4.0
LIN {E6POS: X 1205.139, Y 89.400, Z 531.777, A 35.505, B 81.785, C -144.774, E1 0.000, E2 0.0, E3 0.0, E4 0.0, E5 0.0, E6 0.0} C_DIS
;POWDER FEED RATE  =  3.0
;LASER INTENSITY  =  4.0
LIN {E6POS: X 1203.747, Y 99.560, Z 532.179, A 14.772, B 82.022, C -165.365, E1 0.000, E2 0.0, E3 0.0, E4 0.0, E5 0.0, E6 0.0} C_DIS
;POWDER FEED RATE  =  3.0
;LASER INTENSITY  =  4.0
LIN {E6POS: X 1202.335, Y 109.720, Z 532.237, A 7.934, B 81.732, C -172.148, E1 0.000, E2 0.0, E3 0.0, E4 0.0, E5 0.0, E6 0.0} C_DIS
;POWDER FEED RATE  =  3.0
;LASER INTENSITY  =  4.0
LIN {E6POS: X 1200.919, Y 119.880, Z 532.237, A 7.934, B 81.321, C -172.156, E1 0.000, E2 0.0, E3 0.0, E4 0.0, E5 0.0, E6 0.0} C_DIS
;POWDER FEED RATE  =  3.0
;LASER INTENSITY  =  4.0
LIN {E6POS: X 1199.503, Y 130.040, Z 532.237, A 7.934, B 80.867, C -172.165, E1 0.000, E2 0.0, E3 0.0, E4 0.0, E5 0.0, E6 0.0} C_DIS
;POWDER FEED RATE  =  3.0
;LASER INTENSITY  =  4.0
LIN {E6POS: X 1198.087, Y 140.200, Z 532.237, A 7.934, B 80.363, C -172.177, E1 0.000, E2 0.0, E3 0.0, E4 0.0, E5 0.0, E6 0.0} C_DIS
;POWDER FEED RATE  =  3.0
;LASER INTENSITY  =  4.0
>>>>>>>>>>>>>>>>>>>>>>>>>>>>POWDER FEED OFF  at=START
>>>>>>>>>>>>>>>>>>>>>>>>>>>>LASER OFF at=START
>>>>>>>>>>>>>>>>>>>>>>>>>>>>GAS SUPPLY OFF  at=START
LIN {E6POS: X 1198.087, Y 140.200, Z 532.237, A 7.934, B 80.363, C -172.177, E1 0.000, E2 0.0, E3 0.0, E4 0.0, E5 0.0, E6 0.0} C_DIS
LIN {E6POS: X 1199.503, Y 130.040, Z 532.237, A 7.934, B 80.867, C -172.165, E1 0.000, E2 0.0, E3 0.0, E4 0.0, E5 0.0, E6 0.0} C_DIS
LIN {E6POS: X 1199.503, Y 130.040, Z 532.237, A 7.934, B 80.867, C -172.165, E1 0.000, E2 0.0, E3 0.0, E4 0.0, E5 0.0, E6 0.0} C_DIS
>>>>>>>>>>>>>>>>>>>>>>>>>>>>GAS SUPPLY ON at=END
>>>>>>>>>>>>>>>>>>>>>>>>>>>>POWDER FEED ON at=END
>>>>>>>>>>>>>>>>>>>>>>>>>>>>LASER ON at=END
LIN {E6POS: X 1265.800, Y -12.200, Z 521.408, A -169.621, B 82.629, C 10.295, E1 0.000, E2 0.0, E3 0.0, E4 0.0, E5 0.0, E6 0.0} C_DIS
;POWDER FEED RATE  =  3.0
;LASER INTENSITY  =  4.0
LIN {E6POS: X 1263.735, Y -2.040, Z 521.408, A -166.313, B 82.255, C 13.567, E1 0.000, E2 0.0, E3 0.0, E4 0.0, E5 0.0, E6 0.0} C_DIS
;POWDER FEED RATE  =  3.0
;LASER INTENSITY  =  4.0
LIN {E6POS: X 1260.442, Y 8.120, Z 521.408, A -156.990, B 81.562, C 22.786, E1 0.000, E2 0.0, E3 0.0, E4 0.0, E5 0.0, E6 0.0} C_DIS
;POWDER FEED RATE  =  3.0
;LASER INTENSITY  =  4.0
LIN {E6POS: X 1254.696, Y 18.280, Z 521.408, A -143.998, B 80.222, C 35.604, E1 0.000, E2 0.0, E3 0.0, E4 0.0, E5 0.0, E6 0.0} C_DIS
;POWDER FEED RATE  =  3.0
;LASER INTENSITY  =  4.0
LIN {E6POS: X 1245.888, Y 28.440, Z 521.483, A -141.119, B 79.919, C 38.446, E1 0.000, E2 0.0, E3 0.0, E4 0.0, E5 0.0, E6 0.0} C_DIS
;POWDER FEED RATE  =  3.0
;LASER INTENSITY  =  4.0
LIN {E6POS: X 1235.886, Y 38.600, Z 522.008, A -165.382, B 82.551, C 14.500, E1 0.000, E2 0.0, E3 0.0, E4 0.0, E5 0.0, E6 0.0} C_DIS
;POWDER FEED RATE  =  3.0
;LASER INTENSITY  =  4.0
LIN {E6POS: X 1227.178, Y 48.760, Z 523.435, A 126.019, B 80.769, C -53.625, E1 0.000, E2 0.0, E3 0.0, E4 0.0, E5 0.0, E6 0.0} C_DIS
;POWDER FEED RATE  =  3.0
;LASER INTENSITY  =  4.0
LIN {E6POS: X 1221.620, Y 58.920, Z 525.987, A 98.498, B 74.636, C -81.192, E1 0.000, E2 0.0, E3 0.0, E4 0.0, E5 0.0, E6 0.0} C_DIS
;POWDER FEED RATE  =  3.0
;LASER INTENSITY  =  4.0
LIN {E6POS: X 1218.549, Y 69.080, Z 528.989, A 84.885, B 73.556, C -95.332, E1 0.000, E2 0.0, E3 0.0, E4 0.0, E5 0.0, E6 0.0} C_DIS
;POWDER FEED RATE  =  3.0
;LASER INTENSITY  =  4.0
LIN {E6POS: X 1216.671, Y 79.240, Z 531.541, A 67.857, B 76.982, C -112.669, E1 0.000, E2 0.0, E3 0.0, E4 0.0, E5 0.0, E6 0.0} C_DIS
;POWDER FEED RATE  =  3.0
;LASER INTENSITY  =  4.0
LIN {E6POS: X 1214.916, Y 89.400, Z 532.968, A 41.406, B 80.485, C -138.988, E1 0.000, E2 0.0, E3 0.0, E4 0.0, E5 0.0, E6 0.0} C_DIS
;POWDER FEED RATE  =  3.0
;LASER INTENSITY  =  4.0
LIN {E6POS: X 1213.094, Y 99.560, Z 533.493, A 18.481, B 81.299, C -161.718, E1 0.000, E2 0.0, E3 0.0, E4 0.0, E5 0.0, E6 0.0} C_DIS
;POWDER FEED RATE  =  3.0
;LASER INTENSITY  =  4.0
LIN {E6POS: X 1211.238, Y 109.720, Z 533.568, A 10.379, B 81.066, C -169.745, E1 0.000, E2 0.0, E3 0.0, E4 0.0, E5 0.0, E6 0.0} C_DIS
;POWDER FEED RATE  =  3.0
;LASER INTENSITY  =  4.0
LIN {E6POS: X 1209.378, Y 119.880, Z 533.568, A 10.379, B 80.588, C -169.758, E1 0.000, E2 0.0, E3 0.0, E4 0.0, E5 0.0, E6 0.0} C_DIS
;POWDER FEED RATE  =  3.0
;LASER INTENSITY  =  4.0
LIN {E6POS: X 1207.517, Y 130.040, Z 533.568, A 10.379, B 80.056, C -169.774, E1 0.000, E2 0.0, E3 0.0, E4 0.0, E5 0.0, E6 0.0} C_DIS
;POWDER FEED RATE  =  3.0
;LASER INTENSITY  =  4.0
LIN {E6POS: X 1205.656, Y 140.200, Z 533.568, A 10.379, B 79.461, C -169.793, E1 0.000, E2 0.0, E3 0.0, E4 0.0, E5 0.0, E6 0.0} C_DIS
;POWDER FEED RATE  =  3.0
;LASER INTENSITY  =  4.0
>>>>>>>>>>>>>>>>>>>>>>>>>>>>POWDER FEED OFF  at=START
>>>>>>>>>>>>>>>>>>>>>>>>>>>>LASER OFF at=START
>>>>>>>>>>>>>>>>>>>>>>>>>>>>GAS SUPPLY OFF  at=START
LIN {E6POS: X 1205.656, Y 140.200, Z 533.568, A 10.379, B 79.461, C -169.793, E1 0.000, E2 0.0, E3 0.0, E4 0.0, E5 0.0, E6 0.0} C_DIS
LIN {E6POS: X 1207.517, Y 130.040, Z 533.568, A 10.379, B 80.056, C -169.774, E1 0.000, E2 0.0, E3 0.0, E4 0.0, E5 0.0, E6 0.0} C_DIS
LIN {E6POS: X 1207.517, Y 130.040, Z 533.568, A 10.379, B 80.056, C -169.774, E1 0.000, E2 0.0, E3 0.0, E4 0.0, E5 0.0, E6 0.0} C_DIS
>>>>>>>>>>>>>>>>>>>>>>>>>>>>GAS SUPPLY ON at=END
>>>>>>>>>>>>>>>>>>>>>>>>>>>>POWDER FEED ON at=END
>>>>>>>>>>>>>>>>>>>>>>>>>>>>LASER ON at=END
LIN {E6POS: X 1278.198, Y -12.200, Z 519.817, A -167.011, B 82.455, C 12.881, E1 0.000, E2 0.0, E3 0.0, E4 0.0, E5 0.0, E6 0.0} C_DIS
;POWDER FEED RATE  =  3.0
;LASER INTENSITY  =  4.0
LIN {E6POS: X 1275.663, Y -2.040, Z 519.817, A -163.969, B 82.048, C 15.885, E1 0.000, E2 0.0, E3 0.0, E4 0.0, E5 0.0, E6 0.0} C_DIS
;POWDER FEED RATE  =  3.0
;LASER INTENSITY  =  4.0
LIN {E6POS: X 1271.976, Y 8.120, Z 519.817, A -155.425, B 81.312, C 24.326, E1 0.000, E2 0.0, E3 0.0, E4 0.0, E5 0.0, E6 0.0} C_DIS
;POWDER FEED RATE  =  3.0
;LASER INTENSITY  =  4.0
LIN {E6POS: X 1265.986, Y 18.280, Z 519.817, A -143.476, B 79.977, C 36.103, E1 0.000, E2 0.0, E3 0.0, E4 0.0, E5 0.0, E6 0.0} C_DIS
;POWDER FEED RATE  =  3.0
;LASER INTENSITY  =  4.0
LIN {E6POS: X 1257.127, Y 28.440, Z 519.911, A -142.463, B 79.918, C 37.107, E1 0.000, E2 0.0, E3 0.0, E4 0.0, E5 0.0, E6 0.0} C_DIS
;POWDER FEED RATE  =  3.0
;LASER INTENSITY  =  4.0
LIN {E6POS: X 1247.166, Y 38.600, Z 520.567, A -174.500, B 82.636, C 5.455, E1 0.000, E2 0.0, E3 0.0, E4 0.0, E5 0.0, E6 0.0} C_DIS
;POWDER FEED RATE  =  3.0
;LASER INTENSITY  =  4.0
LIN {E6POS: X 1238.455, Y 48.760, Z 522.350, A 118.231, B 78.461, C -61.279, E1 0.000, E2 0.0, E3 0.0, E4 0.0, E5 0.0, E6 0.0} C_DIS
;POWDER FEED RATE  =  3.0
;LASER INTENSITY  =  4.0
LIN {E6POS: X 1232.746, Y 58.920, Z 525.539, A 96.606, B 70.943, C -83.014, E1 0.000, E2 0.0, E3 0.0, E4 0.0, E5 0.0, E6 0.0} C_DIS
;POWDER FEED RATE  =  3.0
;LASER INTENSITY  =  4.0
LIN {E6POS: X 1229.389, Y 69.080, Z 529.291, A 85.437, B 69.759, C -94.862, E1 0.000, E2 0.0, E3 0.0, E4 0.0, E5 0.0, E6 0.0} C_DIS
;POWDER FEED RATE  =  3.0
;LASER INTENSITY  =  4.0
LIN {E6POS: X 1227.134, Y 79.240, Z 532.480, A 71.063, B 74.152, C -109.629, E1 0.000, E2 0.0, E3 0.0, E4 0.0, E5 0.0, E6 0.0} C_DIS
;POWDER FEED RATE  =  3.0
;LASER INTENSITY  =  4.0
LIN {E6POS: X 1224.948, Y 89.400, Z 534.262, A 46.654, B 79.105, C -133.866, E1 0.000, E2 0.0, E3 0.0, E4 0.0, E5 0.0, E6 0.0} C_DIS
;POWDER FEED RATE  =  3.0
;LASER INTENSITY  =  4.0
LIN {E6POS: X 1222.662, Y 99.560, Z 534.919, A 22.283, B 80.638, C -157.985, E1 0.000, E2 0.0, E3 0.0, E4 0.0, E5 0.0, E6 0.0} C_DIS
;POWDER FEED RATE  =  3.0
;LASER INTENSITY  =  4.0
LIN {E6POS: X 1220.327, Y 109.720, Z 535.013, A 12.989, B 80.508, C -167.183, E1 0.000, E2 0.0, E3 0.0, E4 0.0, E5 0.0, E6 0.0} C_DIS
;POWDER FEED RATE  =  3.0
;LASER INTENSITY  =  4.0
LIN {E6POS: X 1217.983, Y 119.880, Z 535.013, A 12.989, B 79.973, C -167.202, E1 0.000, E2 0.0, E3 0.0, E4 0.0, E5 0.0, E6 0.0} C_DIS
;POWDER FEED RATE  =  3.0
;LASER INTENSITY  =  4.0
LIN {E6POS: X 1215.639, Y 130.040, Z 535.013, A 12.989, B 79.374, C -167.226, E1 0.000, E2 0.0, E3 0.0, E4 0.0, E5 0.0, E6 0.0} C_DIS
;POWDER FEED RATE  =  3.0
;LASER INTENSITY  =  4.0
LIN {E6POS: X 1213.296, Y 140.200, Z 535.013, A 12.989, B 78.699, C -167.254, E1 0.000, E2 0.0, E3 0.0, E4 0.0, E5 0.0, E6 0.0} C_DIS
;POWDER FEED RATE  =  3.0
;LASER INTENSITY  =  4.0
>>>>>>>>>>>>>>>>>>>>>>>>>>>>POWDER FEED OFF  at=START
>>>>>>>>>>>>>>>>>>>>>>>>>>>>LASER OFF at=START
>>>>>>>>>>>>>>>>>>>>>>>>>>>>GAS SUPPLY OFF  at=START
LIN {E6POS: X 1213.296, Y 140.200, Z 535.013, A 12.989, B 78.699, C -167.254, E1 0.000, E2 0.0, E3 0.0, E4 0.0, E5 0.0, E6 0.0} C_DIS
LIN {E6POS: X 1215.639, Y 130.040, Z 535.013, A 12.989, B 79.374, C -167.226, E1 0.000, E2 0.0, E3 0.0, E4 0.0, E5 0.0, E6 0.0} C_DIS
LIN {E6POS: X 1215.639, Y 130.040, Z 535.013, A 12.989, B 79.374, C -167.226, E1 0.000, E2 0.0, E3 0.0, E4 0.0, E5 0.0, E6 0.0} C_DIS
>>>>>>>>>>>>>>>>>>>>>>>>>>>>GAS SUPPLY ON at=END
>>>>>>>>>>>>>>>>>>>>>>>>>>>>POWDER FEED ON at=END
>>>>>>>>>>>>>>>>>>>>>>>>>>>>LASER ON at=END
LIN {E6POS: X 1290.847, Y -12.200, Z 518.184, A -164.298, B 82.376, C 15.570, E1 0.000, E2 0.0, E3 0.0, E4 0.0, E5 0.0, E6 0.0} C_DIS
;POWDER FEED RATE  =  3.0
;LASER INTENSITY  =  4.0
LIN {E6POS: X 1287.813, Y -2.040, Z 518.184, A -161.539, B 81.944, C 18.291, E1 0.000, E2 0.0, E3 0.0, E4 0.0, E5 0.0, E6 0.0} C_DIS
;POWDER FEED RATE  =  3.0
;LASER INTENSITY  =  4.0
LIN {E6POS: X 1283.707, Y 8.120, Z 518.184, A -153.805, B 81.186, C 25.927, E1 0.000, E2 0.0, E3 0.0, E4 0.0, E5 0.0, E6 0.0} C_DIS
;POWDER FEED RATE  =  3.0
;LASER INTENSITY  =  4.0
LIN {E6POS: X 1277.459, Y 18.280, Z 518.184, A -142.929, B 79.887, C 36.640, E1 0.000, E2 0.0, E3 0.0, E4 0.0, E5 0.0, E6 0.0} C_DIS
;POWDER FEED RATE  =  3.0
;LASER INTENSITY  =  4.0
LIN {E6POS: X 1268.546, Y 28.440, Z 518.297, A -144.023, B 80.098, C 35.569, E1 0.000, E2 0.0, E3 0.0, E4 0.0, E5 0.0, E6 0.0} C_DIS
;POWDER FEED RATE  =  3.0
;LASER INTENSITY  =  4.0
LIN {E6POS: X 1258.632, Y 38.600, Z 519.090, A 174.940, B 82.643, C -5.019, E1 0.000, E2 0.0, E3 0.0, E4 0.0, E5 0.0, E6 0.0} C_DIS
;POWDER FEED RATE  =  3.0
;LASER INTENSITY  =  4.0
LIN {E6POS: X 1249.930, Y 48.760, Z 521.244, A 112.451, B 75.917, C -66.925, E1 0.000, E2 0.0, E3 0.0, E4 0.0, E5 0.0, E6 0.0} C_DIS
;POWDER FEED RATE  =  3.0
;LASER INTENSITY  =  4.0
LIN {E6POS: X 1244.082, Y 58.920, Z 525.098, A 95.170, B 67.222, C -84.396, E1 0.000, E2 0.0, E3 0.0, E4 0.0, E5 0.0, E6 0.0} C_DIS
;POWDER FEED RATE  =  3.0
;LASER INTENSITY  =  4.0
LIN {E6POS: X 1240.446, Y 69.080, Z 529.632, A 85.827, B 65.979, C -94.567, E1 0.000, E2 0.0, E3 0.0, E4 0.0, E5 0.0, E6 0.0} C_DIS
;POWDER FEED RATE  =  3.0
;LASER INTENSITY  =  4.0
LIN {E6POS: X 1237.811, Y 79.240, Z 533.486, A 73.523, B 71.263, C -107.345, E1 0.000, E2 0.0, E3 0.0, E4 0.0, E5 0.0, E6 0.0} C_DIS
;POWDER FEED RATE  =  3.0
;LASER INTENSITY  =  4.0
LIN {E6POS: X 1235.178, Y 89.400, Z 535.640, A 51.226, B 77.665, C -129.429, E1 0.000, E2 0.0, E3 0.0, E4 0.0, E5 0.0, E6 0.0} C_DIS
;POWDER FEED RATE  =  3.0
;LASER INTENSITY  =  4.0
LIN {E6POS: X 1232.404, Y 99.560, Z 536.433, A 26.080, B 80.022, C -154.263, E1 0.000, E2 0.0, E3 0.0, E4 0.0, E5 0.0, E6 0.0} C_DIS
;POWDER FEED RATE  =  3.0
;LASER INTENSITY  =  4.0
LIN {E6POS: X 1229.560, Y 109.720, Z 536.547, A 15.702, B 80.042, C -164.523, E1 0.000, E2 0.0, E3 0.0, E4 0.0, E5 0.0, E6 0.0} C_DIS
;POWDER FEED RATE  =  3.0
;LASER INTENSITY  =  4.0
LIN {E6POS: X 1226.703, Y 119.880, Z 536.547, A 15.702, B 79.459, C -164.550, E1 0.000, E2 0.0, E3 0.0, E4 0.0, E5 0.0, E6 0.0} C_DIS
;POWDER FEED RATE  =  3.0
;LASER INTENSITY  =  4.0
LIN {E6POS: X 1223.847, Y 130.040, Z 536.547, A 15.702, B 78.804, C -164.582, E1 0.000, E2 0.0, E3 0.0, E4 0.0, E5 0.0, E6 0.0} C_DIS
;POWDER FEED RATE  =  3.0
;LASER INTENSITY  =  4.0
LIN {E6POS: X 1220.991, Y 140.200, Z 536.547, A 15.702, B 78.064, C -164.621, E1 0.000, E2 0.0, E3 0.0, E4 0.0, E5 0.0, E6 0.0} C_DIS
;POWDER FEED RATE  =  3.0
;LASER INTENSITY  =  4.0
>>>>>>>>>>>>>>>>>>>>>>>>>>>>POWDER FEED OFF  at=START
>>>>>>>>>>>>>>>>>>>>>>>>>>>>LASER OFF at=START
>>>>>>>>>>>>>>>>>>>>>>>>>>>>GAS SUPPLY OFF  at=START
LIN {E6POS: X 1220.991, Y 140.200, Z 536.547, A 15.702, B 78.064, C -164.621, E1 0.000, E2 0.0, E3 0.0, E4 0.0, E5 0.0, E6 0.0} C_DIS
LIN {E6POS: X 1223.847, Y 130.040, Z 536.547, A 15.702, B 78.804, C -164.582, E1 0.000, E2 0.0, E3 0.0, E4 0.0, E5 0.0, E6 0.0} C_DIS
LIN {E6POS: X 1223.847, Y 130.040, Z 536.547, A 15.702, B 78.804, C -164.582, E1 0.000, E2 0.0, E3 0.0, E4 0.0, E5 0.0, E6 0.0} C_DIS
>>>>>>>>>>>>>>>>>>>>>>>>>>>>GAS SUPPLY ON at=END
>>>>>>>>>>>>>>>>>>>>>>>>>>>>POWDER FEED ON at=END
>>>>>>>>>>>>>>>>>>>>>>>>>>>>LASER ON at=END
LIN {E6POS: X 1303.630, Y -12.200, Z 516.548, A -161.545, B 82.390, C 18.304, E1 0.000, E2 0.0, E3 0.0, E4 0.0, E5 0.0, E6 0.0} C_DIS
;POWDER FEED RATE  =  3.0
;LASER INTENSITY  =  4.0
LIN {E6POS: X 1300.075, Y -2.040, Z 516.548, A -159.077, B 81.945, C 20.734, E1 0.000, E2 0.0, E3 0.0, E4 0.0, E5 0.0, E6 0.0} C_DIS
;POWDER FEED RATE  =  3.0
;LASER INTENSITY  =  4.0
LIN {E6POS: X 1295.532, Y 8.120, Z 516.548, A -152.163, B 81.185, C 27.557, E1 0.000, E2 0.0, E3 0.0, E4 0.0, E5 0.0, E6 0.0} C_DIS
;POWDER FEED RATE  =  3.0
;LASER INTENSITY  =  4.0
LIN {E6POS: X 1289.015, Y 18.280, Z 516.548, A -142.368, B 79.949, C 37.204, E1 0.000, E2 0.0, E3 0.0, E4 0.0, E5 0.0, E6 0.0} C_DIS
;POWDER FEED RATE  =  3.0
;LASER INTENSITY  =  4.0
LIN {E6POS: X 1280.046, Y 28.440, Z 516.681, A -145.862, B 80.446, C 33.767, E1 0.000, E2 0.0, E3 0.0, E4 0.0, E5 0.0, E6 0.0} C_DIS
;POWDER FEED RATE  =  3.0
;LASER INTENSITY  =  4.0
LIN {E6POS: X 1270.187, Y 38.600, Z 517.615, A 163.374, B 82.480, C -16.491, E1 0.000, E2 0.0, E3 0.0, E4 0.0, E5 0.0, E6 0.0} C_DIS
;POWDER FEED RATE  =  3.0
;LASER INTENSITY  =  4.0
LIN {E6POS: X 1261.508, Y 48.760, Z 520.148, A 108.050, B 73.239, C -71.204, E1 0.000, E2 0.0, E3 0.0, E4 0.0, E5 0.0, E6 0.0} C_DIS
;POWDER FEED RATE  =  3.0
;LASER INTENSITY  =  4.0
LIN {E6POS: X 1255.539, Y 58.920, Z 524.681, A 94.028, B 63.586, C -85.505, E1 0.000, E2 0.0, E3 0.0, E4 0.0, E5 0.0, E6 0.0} C_DIS
;POWDER FEED RATE  =  3.0
;LASER INTENSITY  =  4.0
LIN {E6POS: X 1251.642, Y 69.080, Z 530.013, A 86.100, B 62.328, C -94.401, E1 0.000, E2 0.0, E3 0.0, E4 0.0, E5 0.0, E6 0.0} C_DIS
;POWDER FEED RATE  =  3.0
;LASER INTENSITY  =  4.0
LIN {E6POS: X 1248.635, Y 79.240, Z 534.546, A 75.444, B 68.399, C -105.604, E1 0.000, E2 0.0, E3 0.0, E4 0.0, E5 0.0, E6 0.0} C_DIS
;POWDER FEED RATE  =  3.0
;LASER INTENSITY  =  4.0
LIN {E6POS: X 1245.550, Y 89.400, Z 537.079, A 55.160, B 76.198, C -125.631, E1 0.000, E2 0.0, E3 0.0, E4 0.0, E5 0.0, E6 0.0} C_DIS
;POWDER FEED RATE  =  3.0
;LASER INTENSITY  =  4.0
LIN {E6POS: X 1242.273, Y 99.560, Z 538.012, A 29.788, B 79.446, C -150.632, E1 0.000, E2 0.0, E3 0.0, E4 0.0, E5 0.0, E6 0.0} C_DIS
;POWDER FEED RATE  =  3.0
;LASER INTENSITY  =  4.0
LIN {E6POS: X 1238.898, Y 109.720, Z 538.146, A 18.455, B 79.658, C -161.825, E1 0.000, E2 0.0, E3 0.0, E4 0.0, E5 0.0, E6 0.0} C_DIS
;POWDER FEED RATE  =  3.0
;LASER INTENSITY  =  4.0
LIN {E6POS: X 1235.507, Y 119.880, Z 538.146, A 18.455, B 79.038, C -161.859, E1 0.000, E2 0.0, E3 0.0, E4 0.0, E5 0.0, E6 0.0} C_DIS
;POWDER FEED RATE  =  3.0
;LASER INTENSITY  =  4.0
LIN {E6POS: X 1232.117, Y 130.040, Z 538.146, A 18.455, B 78.340, C -161.900, E1 0.000, E2 0.0, E3 0.0, E4 0.0, E5 0.0, E6 0.0} C_DIS
;POWDER FEED RATE  =  3.0
;LASER INTENSITY  =  4.0
LIN {E6POS: X 1228.726, Y 140.200, Z 538.146, A 18.455, B 77.549, C -161.950, E1 0.000, E2 0.0, E3 0.0, E4 0.0, E5 0.0, E6 0.0} C_DIS
;POWDER FEED RATE  =  3.0
;LASER INTENSITY  =  4.0
>>>>>>>>>>>>>>>>>>>>>>>>>>>>POWDER FEED OFF  at=START
>>>>>>>>>>>>>>>>>>>>>>>>>>>>LASER OFF at=START
>>>>>>>>>>>>>>>>>>>>>>>>>>>>GAS SUPPLY OFF  at=START
LIN {E6POS: X 1228.726, Y 140.200, Z 538.146, A 18.455, B 77.549, C -161.950, E1 0.000, E2 0.0, E3 0.0, E4 0.0, E5 0.0, E6 0.0} C_DIS
LIN {E6POS: X 1232.117, Y 130.040, Z 538.146, A 18.455, B 78.340, C -161.900, E1 0.000, E2 0.0, E3 0.0, E4 0.0, E5 0.0, E6 0.0} C_DIS
LIN {E6POS: X 1232.117, Y 130.040, Z 538.146, A 18.455, B 78.340, C -161.900, E1 0.000, E2 0.0, E3 0.0, E4 0.0, E5 0.0, E6 0.0} C_DIS
>>>>>>>>>>>>>>>>>>>>>>>>>>>>GAS SUPPLY ON at=END
>>>>>>>>>>>>>>>>>>>>>>>>>>>>POWDER FEED ON at=END
>>>>>>>>>>>>>>>>>>>>>>>>>>>>LASER ON at=END
LIN {E6POS: X 1316.427, Y -12.200, Z 514.950, A -158.811, B 82.506, C 21.024, E1 0.000, E2 0.0, E3 0.0, E4 0.0, E5 0.0, E6 0.0} C_DIS
;POWDER FEED RATE  =  3.0
;LASER INTENSITY  =  4.0
LIN {E6POS: X 1312.338, Y -2.040, Z 514.950, A -156.635, B 82.060, C 23.165, E1 0.000, E2 0.0, E3 0.0, E4 0.0, E5 0.0, E6 0.0} C_DIS
;POWDER FEED RATE  =  3.0
;LASER INTENSITY  =  4.0
LIN {E6POS: X 1307.348, Y 8.120, Z 514.950, A -150.529, B 81.318, C 29.189, E1 0.000, E2 0.0, E3 0.0, E4 0.0, E5 0.0, E6 0.0} C_DIS
;POWDER FEED RATE  =  3.0
;LASER INTENSITY  =  4.0
LIN {E6POS: X 1300.555, Y 18.280, Z 514.950, A -141.801, B 80.171, C 37.788, E1 0.000, E2 0.0, E3 0.0, E4 0.0, E5 0.0, E6 0.0} C_DIS
;POWDER FEED RATE  =  3.0
;LASER INTENSITY  =  4.0
LIN {E6POS: X 1291.529, Y 28.440, Z 515.104, A -148.080, B 80.957, C 31.599, E1 0.000, E2 0.0, E3 0.0, E4 0.0, E5 0.0, E6 0.0} C_DIS
;POWDER FEED RATE  =  3.0
;LASER INTENSITY  =  4.0
LIN {E6POS: X 1281.732, Y 38.600, Z 516.177, A 151.531, B 82.084, C -28.239, E1 0.000, E2 0.0, E3 0.0, E4 0.0, E5 0.0, E6 0.0} C_DIS
;POWDER FEED RATE  =  3.0
;LASER INTENSITY  =  4.0
LIN {E6POS: X 1273.093, Y 48.760, Z 519.090, A 104.581, B 70.517, C -74.574, E1 0.000, E2 0.0, E3 0.0, E4 0.0, E5 0.0, E6 0.0} C_DIS
;POWDER FEED RATE  =  3.0
;LASER INTENSITY  =  4.0
LIN {E6POS: X 1267.029, Y 58.920, Z 524.302, A 93.079, B 60.127, C -86.451, E1 0.000, E2 0.0, E3 0.0, E4 0.0, E5 0.0, E6 0.0} C_DIS
;POWDER FEED RATE  =  3.0
;LASER INTENSITY  =  4.0
LIN {E6POS: X 1262.898, Y 69.080, Z 530.434, A 86.285, B 58.893, C -94.337, E1 0.000, E2 0.0, E3 0.0, E4 0.0, E5 0.0, E6 0.0} C_DIS
;POWDER FEED RATE  =  3.0
;LASER INTENSITY  =  4.0
LIN {E6POS: X 1259.539, Y 79.240, Z 535.646, A 76.965, B 65.637, C -104.259, E1 0.000, E2 0.0, E3 0.0, E4 0.0, E5 0.0, E6 0.0} C_DIS
;POWDER FEED RATE  =  3.0
;LASER INTENSITY  =  4.0
LIN {E6POS: X 1256.008, Y 89.400, Z 538.559, A 58.527, B 74.741, C -122.396, E1 0.000, E2 0.0, E3 0.0, E4 0.0, E5 0.0, E6 0.0} C_DIS
;POWDER FEED RATE  =  3.0
;LASER INTENSITY  =  4.0
LIN {E6POS: X 1252.219, Y 99.560, Z 539.632, A 33.340, B 78.915, C -147.153, E1 0.000, E2 0.0, E3 0.0, E4 0.0, E5 0.0, E6 0.0} C_DIS
;POWDER FEED RATE  =  3.0
;LASER INTENSITY  =  4.0
LIN {E6POS: X 1248.302, Y 109.720, Z 539.785, A 21.189, B 79.354, C -159.144, E1 0.000, E2 0.0, E3 0.0, E4 0.0, E5 0.0, E6 0.0} C_DIS
;POWDER FEED RATE  =  3.0
;LASER INTENSITY  =  4.0
LIN {E6POS: X 1244.364, Y 119.880, Z 539.785, A 21.189, B 78.708, C -159.185, E1 0.000, E2 0.0, E3 0.0, E4 0.0, E5 0.0, E6 0.0} C_DIS
;POWDER FEED RATE  =  3.0
;LASER INTENSITY  =  4.0
LIN {E6POS: X 1240.425, Y 130.040, Z 539.785, A 21.189, B 77.980, C -159.235, E1 0.000, E2 0.0, E3 0.0, E4 0.0, E5 0.0, E6 0.0} C_DIS
;POWDER FEED RATE  =  3.0
;LASER INTENSITY  =  4.0
LIN {E6POS: X 1236.486, Y 140.200, Z 539.785, A 21.189, B 77.153, C -159.296, E1 0.000, E2 0.0, E3 0.0, E4 0.0, E5 0.0, E6 0.0} C_DIS
;POWDER FEED RATE  =  3.0
;LASER INTENSITY  =  4.0
>>>>>>>>>>>>>>>>>>>>>>>>>>>>POWDER FEED OFF  at=START
>>>>>>>>>>>>>>>>>>>>>>>>>>>>LASER OFF at=START
>>>>>>>>>>>>>>>>>>>>>>>>>>>>GAS SUPPLY OFF  at=START
LIN {E6POS: X 1236.486, Y 140.200, Z 539.785, A 21.189, B 77.153, C -159.296, E1 0.000, E2 0.0, E3 0.0, E4 0.0, E5 0.0, E6 0.0} C_DIS
LIN {E6POS: X 1240.425, Y 130.040, Z 539.785, A 21.189, B 77.980, C -159.235, E1 0.000, E2 0.0, E3 0.0, E4 0.0, E5 0.0, E6 0.0} C_DIS
LIN {E6POS: X 1240.425, Y 130.040, Z 539.785, A 21.189, B 77.980, C -159.235, E1 0.000, E2 0.0, E3 0.0, E4 0.0, E5 0.0, E6 0.0} C_DIS
>>>>>>>>>>>>>>>>>>>>>>>>>>>>GAS SUPPLY ON at=END
>>>>>>>>>>>>>>>>>>>>>>>>>>>>POWDER FEED ON at=END
>>>>>>>>>>>>>>>>>>>>>>>>>>>>LASER ON at=END
LIN {E6POS: X 1329.120, Y -12.200, Z 513.430, A -156.149, B 82.743, C 23.681, E1 0.000, E2 0.0, E3 0.0, E4 0.0, E5 0.0, E6 0.0} C_DIS
;POWDER FEED RATE  =  3.0
;LASER INTENSITY  =  4.0
LIN {E6POS: X 1324.492, Y -2.040, Z 513.430, A -154.256, B 82.307, C 25.542, E1 0.000, E2 0.0, E3 0.0, E4 0.0, E5 0.0, E6 0.0} C_DIS
;POWDER FEED RATE  =  3.0
;LASER INTENSITY  =  4.0
LIN {E6POS: X 1319.049, Y 8.120, Z 513.430, A -148.931, B 81.605, C 30.797, E1 0.000, E2 0.0, E3 0.0, E4 0.0, E5 0.0, E6 0.0} C_DIS
;POWDER FEED RATE  =  3.0
;LASER INTENSITY  =  4.0
LIN {E6POS: X 1311.978, Y 18.280, Z 513.430, A -141.237, B 80.569, C 38.383, E1 0.000, E2 0.0, E3 0.0, E4 0.0, E5 0.0, E6 0.0} C_DIS
;POWDER FEED RATE  =  3.0
;LASER INTENSITY  =  4.0
LIN {E6POS: X 1302.897, Y 28.440, Z 513.603, A -150.854, B 81.634, C 28.885, E1 0.000, E2 0.0, E3 0.0, E4 0.0, E5 0.0, E6 0.0} C_DIS
;POWDER FEED RATE  =  3.0
;LASER INTENSITY  =  4.0
LIN {E6POS: X 1293.168, Y 38.600, Z 514.814, A 140.163, B 81.430, C -39.521, E1 0.000, E2 0.0, E3 0.0, E4 0.0, E5 0.0, E6 0.0} C_DIS
;POWDER FEED RATE  =  3.0
;LASER INTENSITY  =  4.0
LIN {E6POS: X 1284.589, Y 48.760, Z 518.099, A 101.741, B 67.826, C -77.351, E1 0.000, E2 0.0, E3 0.0, E4 0.0, E5 0.0, E6 0.0} C_DIS
;POWDER FEED RATE  =  3.0
;LASER INTENSITY  =  4.0
LIN {E6POS: X 1278.465, Y 58.920, Z 523.978, A 92.254, B 56.915, C -87.310, E1 0.000, E2 0.0, E3 0.0, E4 0.0, E5 0.0, E6 0.0} C_DIS
;POWDER FEED RATE  =  3.0
;LASER INTENSITY  =  4.0
LIN {E6POS: X 1274.137, Y 69.080, Z 530.894, A 86.397, B 55.740, C -94.357, E1 0.000, E2 0.0, E3 0.0, E4 0.0, E5 0.0, E6 0.0} C_DIS
;POWDER FEED RATE  =  3.0
;LASER INTENSITY  =  4.0
LIN {E6POS: X 1270.457, Y 79.240, Z 536.773, A 78.187, B 63.043, C -103.206, E1 0.000, E2 0.0, E3 0.0, E4 0.0, E5 0.0, E6 0.0} C_DIS
;POWDER FEED RATE  =  3.0
;LASER INTENSITY  =  4.0
LIN {E6POS: X 1266.494, Y 89.400, Z 540.058, A 61.409, B 73.335, C -119.636, E1 0.000, E2 0.0, E3 0.0, E4 0.0, E5 0.0, E6 0.0} C_DIS
;POWDER FEED RATE  =  3.0
;LASER INTENSITY  =  4.0
LIN {E6POS: X 1262.197, Y 99.560, Z 541.268, A 36.692, B 78.439, C -143.869, E1 0.000, E2 0.0, E3 0.0, E4 0.0, E5 0.0, E6 0.0} C_DIS
;POWDER FEED RATE  =  3.0
;LASER INTENSITY  =  4.0
LIN {E6POS: X 1257.733, Y 109.720, Z 541.441, A 23.851, B 79.133, C -156.530, E1 0.000, E2 0.0, E3 0.0, E4 0.0, E5 0.0, E6 0.0} C_DIS
;POWDER FEED RATE  =  3.0
;LASER INTENSITY  =  4.0
LIN {E6POS: X 1253.241, Y 119.880, Z 541.441, A 23.851, B 78.473, C -156.577, E1 0.000, E2 0.0, E3 0.0, E4 0.0, E5 0.0, E6 0.0} C_DIS
;POWDER FEED RATE  =  3.0
;LASER INTENSITY  =  4.0
LIN {E6POS: X 1248.749, Y 130.040, Z 541.441, A 23.851, B 77.730, C -156.635, E1 0.000, E2 0.0, E3 0.0, E4 0.0, E5 0.0, E6 0.0} C_DIS
;POWDER FEED RATE  =  3.0
;LASER INTENSITY  =  4.0
LIN {E6POS: X 1244.257, Y 140.200, Z 541.441, A 23.851, B 76.885, C -156.704, E1 0.000, E2 0.0, E3 0.0, E4 0.0, E5 0.0, E6 0.0} C_DIS
;POWDER FEED RATE  =  3.0
;LASER INTENSITY  =  4.0
>>>>>>>>>>>>>>>>>>>>>>>>>>>>POWDER FEED OFF  at=START
>>>>>>>>>>>>>>>>>>>>>>>>>>>>LASER OFF at=START
>>>>>>>>>>>>>>>>>>>>>>>>>>>>GAS SUPPLY OFF  at=START
LIN {E6POS: X 1244.257, Y 140.200, Z 541.441, A 23.851, B 76.885, C -156.704, E1 0.000, E2 0.0, E3 0.0, E4 0.0, E5 0.0, E6 0.0} C_DIS
LIN {E6POS: X 1248.749, Y 130.040, Z 541.441, A 23.851, B 77.730, C -156.635, E1 0.000, E2 0.0, E3 0.0, E4 0.0, E5 0.0, E6 0.0} C_DIS
LIN {E6POS: X 1248.749, Y 130.040, Z 541.441, A 23.851, B 77.730, C -156.635, E1 0.000, E2 0.0, E3 0.0, E4 0.0, E5 0.0, E6 0.0} C_DIS
>>>>>>>>>>>>>>>>>>>>>>>>>>>>GAS SUPPLY ON at=END
>>>>>>>>>>>>>>>>>>>>>>>>>>>>POWDER FEED ON at=END
>>>>>>>>>>>>>>>>>>>>>>>>>>>>LASER ON at=END
LIN {E6POS: X 1341.590, Y -12.200, Z 512.028, A -153.604, B 83.129, C 26.232, E1 0.000, E2 0.0, E3 0.0, E4 0.0, E5 0.0, E6 0.0} C_DIS
;POWDER FEED RATE  =  3.0
;LASER INTENSITY  =  4.0
LIN {E6POS: X 1336.426, Y -2.040, Z 512.028, A -151.980, B 82.717, C 27.828, E1 0.000, E2 0.0, E3 0.0, E4 0.0, E5 0.0, E6 0.0} C_DIS
;POWDER FEED RATE  =  3.0
;LASER INTENSITY  =  4.0
LIN {E6POS: X 1330.534, Y 8.120, Z 512.028, A -147.392, B 82.075, C 32.358, E1 0.000, E2 0.0, E3 0.0, E4 0.0, E5 0.0, E6 0.0} C_DIS
;POWDER FEED RATE  =  3.0
;LASER INTENSITY  =  4.0
LIN {E6POS: X 1323.184, Y 18.280, Z 512.028, A -140.684, B 81.170, C 38.981, E1 0.000, E2 0.0, E3 0.0, E4 0.0, E5 0.0, E6 0.0} C_DIS
;POWDER FEED RATE  =  3.0
;LASER INTENSITY  =  4.0
LIN {E6POS: X 1314.050, Y 28.440, Z 512.220, A -154.521, B 82.484, C 25.288, E1 0.000, E2 0.0, E3 0.0, E4 0.0, E5 0.0, E6 0.0} C_DIS
;POWDER FEED RATE  =  3.0
;LASER INTENSITY  =  4.0
LIN {E6POS: X 1304.399, Y 38.600, Z 513.562, A 129.749, B 80.529, C -49.864, E1 0.000, E2 0.0, E3 0.0, E4 0.0, E5 0.0, E6 0.0} C_DIS
;POWDER FEED RATE  =  3.0
;LASER INTENSITY  =  4.0
LIN {E6POS: X 1295.901, Y 48.760, Z 517.205, A 99.314, B 65.228, C -79.761, E1 0.000, E2 0.0, E3 0.0, E4 0.0, E5 0.0, E6 0.0} C_DIS
;POWDER FEED RATE  =  3.0
;LASER INTENSITY  =  4.0
LIN {E6POS: X 1289.757, Y 58.920, Z 523.724, A 91.503, B 53.997, C -88.142, E1 0.000, E2 0.0, E3 0.0, E4 0.0, E5 0.0, E6 0.0} C_DIS
;POWDER FEED RATE  =  3.0
;LASER INTENSITY  =  4.0
LIN {E6POS: X 1285.281, Y 69.080, Z 531.393, A 86.445, B 52.911, C -94.453, E1 0.000, E2 0.0, E3 0.0, E4 0.0, E5 0.0, E6 0.0} C_DIS
;POWDER FEED RATE  =  3.0
;LASER INTENSITY  =  4.0
LIN {E6POS: X 1281.322, Y 79.240, Z 537.912, A 79.178, B 60.666, C -102.368, E1 0.000, E2 0.0, E3 0.0, E4 0.0, E5 0.0, E6 0.0} C_DIS
;POWDER FEED RATE  =  3.0
;LASER INTENSITY  =  4.0
LIN {E6POS: X 1276.952, Y 89.400, Z 541.555, A 63.886, B 72.022, C -117.265, E1 0.000, E2 0.0, E3 0.0, E4 0.0, E5 0.0, E6 0.0} C_DIS
;POWDER FEED RATE  =  3.0
;LASER INTENSITY  =  4.0
LIN {E6POS: X 1272.158, Y 99.560, Z 542.897, A 39.818, B 78.036, C -140.800, E1 0.000, E2 0.0, E3 0.0, E4 0.0, E5 0.0, E6 0.0} C_DIS
;POWDER FEED RATE  =  3.0
;LASER INTENSITY  =  4.0
LIN {E6POS: X 1267.150, Y 109.720, Z 543.089, A 26.396, B 79.005, C -154.024, E1 0.000, E2 0.0, E3 0.0, E4 0.0, E5 0.0, E6 0.0} C_DIS
;POWDER FEED RATE  =  3.0
;LASER INTENSITY  =  4.0
LIN {E6POS: X 1262.108, Y 119.880, Z 543.089, A 26.396, B 78.344, C -154.076, E1 0.000, E2 0.0, E3 0.0, E4 0.0, E5 0.0, E6 0.0} C_DIS
;POWDER FEED RATE  =  3.0
;LASER INTENSITY  =  4.0
LIN {E6POS: X 1257.065, Y 130.040, Z 543.089, A 26.396, B 77.600, C -154.139, E1 0.000, E2 0.0, E3 0.0, E4 0.0, E5 0.0, E6 0.0} C_DIS
;POWDER FEED RATE  =  3.0
;LASER INTENSITY  =  4.0
LIN {E6POS: X 1252.023, Y 140.200, Z 543.089, A 26.396, B 76.756, C -154.214, E1 0.000, E2 0.0, E3 0.0, E4 0.0, E5 0.0, E6 0.0} C_DIS
;POWDER FEED RATE  =  3.0
;LASER INTENSITY  =  4.0
>>>>>>>>>>>>>>>>>>>>>>>>>>>>POWDER FEED OFF  at=START
>>>>>>>>>>>>>>>>>>>>>>>>>>>>LASER OFF at=START
>>>>>>>>>>>>>>>>>>>>>>>>>>>>GAS SUPPLY OFF  at=START
LIN {E6POS: X 1252.023, Y 140.200, Z 543.089, A 26.396, B 76.756, C -154.214, E1 0.000, E2 0.0, E3 0.0, E4 0.0, E5 0.0, E6 0.0} C_DIS
LIN {E6POS: X 1257.065, Y 130.040, Z 543.089, A 26.396, B 77.600, C -154.139, E1 0.000, E2 0.0, E3 0.0, E4 0.0, E5 0.0, E6 0.0} C_DIS
LIN {E6POS: X 1257.065, Y 130.040, Z 543.089, A 26.396, B 77.600, C -154.139, E1 0.000, E2 0.0, E3 0.0, E4 0.0, E5 0.0, E6 0.0} C_DIS
>>>>>>>>>>>>>>>>>>>>>>>>>>>>GAS SUPPLY ON at=END
>>>>>>>>>>>>>>>>>>>>>>>>>>>>POWDER FEED ON at=END
>>>>>>>>>>>>>>>>>>>>>>>>>>>>LASER ON at=END
LIN {E6POS: X 1353.720, Y -12.200, Z 510.784, A -151.213, B 83.707, C 28.641, E1 0.000, E2 0.0, E3 0.0, E4 0.0, E5 0.0, E6 0.0} C_DIS
;POWDER FEED RATE  =  3.0
;LASER INTENSITY  =  4.0
LIN {E6POS: X 1348.030, Y -2.040, Z 510.784, A -149.838, B 83.335, C 29.994, E1 0.000, E2 0.0, E3 0.0, E4 0.0, E5 0.0, E6 0.0} C_DIS
;POWDER FEED RATE  =  3.0
;LASER INTENSITY  =  4.0
LIN {E6POS: X 1341.697, Y 8.120, Z 510.784, A -145.934, B 82.774, C 33.855, E1 0.000, E2 0.0, E3 0.0, E4 0.0, E5 0.0, E6 0.0} C_DIS
;POWDER FEED RATE  =  3.0
;LASER INTENSITY  =  4.0
LIN {E6POS: X 1334.076, Y 18.280, Z 510.784, A -140.151, B 82.017, C 39.575, E1 0.000, E2 0.0, E3 0.0, E4 0.0, E5 0.0, E6 0.0} C_DIS
;POWDER FEED RATE  =  3.0
;LASER INTENSITY  =  4.0
LIN {E6POS: X 1324.889, Y 28.440, Z 510.993, A -159.785, B 83.520, C 20.096, E1 0.000, E2 0.0, E3 0.0, E4 0.0, E5 0.0, E6 0.0} C_DIS
;POWDER FEED RATE  =  3.0
;LASER INTENSITY  =  4.0
LIN {E6POS: X 1315.324, Y 38.600, Z 512.459, A 120.412, B 79.409, C -59.156, E1 0.000, E2 0.0, E3 0.0, E4 0.0, E5 0.0, E6 0.0} C_DIS
;POWDER FEED RATE  =  3.0
;LASER INTENSITY  =  4.0
LIN {E6POS: X 1306.934, Y 48.760, Z 516.437, A 97.143, B 62.772, C -81.978, E1 0.000, E2 0.0, E3 0.0, E4 0.0, E5 0.0, E6 0.0} C_DIS
;POWDER FEED RATE  =  3.0
;LASER INTENSITY  =  4.0
LIN {E6POS: X 1300.817, Y 58.920, Z 523.556, A 90.784, B 51.400, C -88.997, E1 0.000, E2 0.0, E3 0.0, E4 0.0, E5 0.0, E6 0.0} C_DIS
;POWDER FEED RATE  =  3.0
;LASER INTENSITY  =  4.0
LIN {E6POS: X 1296.253, Y 69.080, Z 531.932, A 86.435, B 50.427, C -94.621, E1 0.000, E2 0.0, E3 0.0, E4 0.0, E5 0.0, E6 0.0} C_DIS
;POWDER FEED RATE  =  3.0
;LASER INTENSITY  =  4.0
LIN {E6POS: X 1292.068, Y 79.240, Z 539.051, A 79.991, B 58.548, C -101.689, E1 0.000, E2 0.0, E3 0.0, E4 0.0, E5 0.0, E6 0.0} C_DIS
;POWDER FEED RATE  =  3.0
;LASER INTENSITY  =  4.0
LIN {E6POS: X 1287.326, Y 89.400, Z 543.029, A 66.033, B 70.842, C -115.202, E1 0.000, E2 0.0, E3 0.0, E4 0.0, E5 0.0, E6 0.0} C_DIS
;POWDER FEED RATE  =  3.0
;LASER INTENSITY  =  4.0
LIN {E6POS: X 1282.053, Y 99.560, Z 544.495, A 42.713, B 77.728, C -137.946, E1 0.000, E2 0.0, E3 0.0, E4 0.0, E5 0.0, E6 0.0} C_DIS
;POWDER FEED RATE  =  3.0
;LASER INTENSITY  =  4.0
LIN {E6POS: X 1276.515, Y 109.720, Z 544.704, A 28.787, B 78.985, C -151.661, E1 0.000, E2 0.0, E3 0.0, E4 0.0, E5 0.0, E6 0.0} C_DIS
;POWDER FEED RATE  =  3.0
;LASER INTENSITY  =  4.0
LIN {E6POS: X 1270.933, Y 119.880, Z 544.704, A 28.787, B 78.337, C -151.715, E1 0.000, E2 0.0, E3 0.0, E4 0.0, E5 0.0, E6 0.0} C_DIS
;POWDER FEED RATE  =  3.0
;LASER INTENSITY  =  4.0
LIN {E6POS: X 1265.350, Y 130.040, Z 544.704, A 28.787, B 77.609, C -151.780, E1 0.000, E2 0.0, E3 0.0, E4 0.0, E5 0.0, E6 0.0} C_DIS
;POWDER FEED RATE  =  3.0
;LASER INTENSITY  =  4.0
LIN {E6POS: X 1259.768, Y 140.200, Z 544.704, A 28.787, B 76.786, C -151.858, E1 0.000, E2 0.0, E3 0.0, E4 0.0, E5 0.0, E6 0.0} C_DIS
;POWDER FEED RATE  =  3.0
;LASER INTENSITY  =  4.0
>>>>>>>>>>>>>>>>>>>>>>>>>>>>POWDER FEED OFF  at=START
>>>>>>>>>>>>>>>>>>>>>>>>>>>>LASER OFF at=START
>>>>>>>>>>>>>>>>>>>>>>>>>>>>GAS SUPPLY OFF  at=START
LIN {E6POS: X 1259.768, Y 140.200, Z 544.704, A 28.787, B 76.786, C -151.858, E1 0.000, E2 0.0, E3 0.0, E4 0.0, E5 0.0, E6 0.0} C_DIS
LIN {E6POS: X 1265.350, Y 130.040, Z 544.704, A 28.787, B 77.609, C -151.780, E1 0.000, E2 0.0, E3 0.0, E4 0.0, E5 0.0, E6 0.0} C_DIS
LIN {E6POS: X 1265.350, Y 130.040, Z 544.704, A 28.787, B 77.609, C -151.780, E1 0.000, E2 0.0, E3 0.0, E4 0.0, E5 0.0, E6 0.0} C_DIS
>>>>>>>>>>>>>>>>>>>>>>>>>>>>GAS SUPPLY ON at=END
>>>>>>>>>>>>>>>>>>>>>>>>>>>>POWDER FEED ON at=END
>>>>>>>>>>>>>>>>>>>>>>>>>>>>LASER ON at=END
LIN {E6POS: X 1365.391, Y -12.200, Z 509.738, A -149.006, B 84.541, C 30.879, E1 0.000, E2 0.0, E3 0.0, E4 0.0, E5 0.0, E6 0.0} C_DIS
;POWDER FEED RATE  =  3.0
;LASER INTENSITY  =  4.0
LIN {E6POS: X 1359.194, Y -2.040, Z 509.738, A -147.856, B 84.224, C 32.013, E1 0.000, E2 0.0, E3 0.0, E4 0.0, E5 0.0, E6 0.0} C_DIS
;POWDER FEED RATE  =  3.0
;LASER INTENSITY  =  4.0
LIN {E6POS: X 1352.435, Y 8.120, Z 509.738, A -144.572, B 83.764, C 35.267, E1 0.000, E2 0.0, E3 0.0, E4 0.0, E5 0.0, E6 0.0} C_DIS
;POWDER FEED RATE  =  3.0
;LASER INTENSITY  =  4.0
LIN {E6POS: X 1344.551, Y 18.280, Z 509.738, A -139.644, B 83.170, C 40.155, E1 0.000, E2 0.0, E3 0.0, E4 0.0, E5 0.0, E6 0.0} C_DIS
;POWDER FEED RATE  =  3.0
;LASER INTENSITY  =  4.0
LIN {E6POS: X 1335.316, Y 28.440, Z 509.963, A -168.346, B 84.738, C 11.607, E1 0.000, E2 0.0, E3 0.0, E4 0.0, E5 0.0, E6 0.0} C_DIS
;POWDER FEED RATE  =  3.0
;LASER INTENSITY  =  4.0
LIN {E6POS: X 1325.846, Y 38.600, Z 511.541, A 112.008, B 78.094, C -67.555, E1 0.000, E2 0.0, E3 0.0, E4 0.0, E5 0.0, E6 0.0} C_DIS
;POWDER FEED RATE  =  3.0
;LASER INTENSITY  =  4.0
LIN {E6POS: X 1317.590, Y 48.760, Z 515.825, A 95.097, B 60.493, C -84.148, E1 0.000, E2 0.0, E3 0.0, E4 0.0, E5 0.0, E6 0.0} C_DIS
;POWDER FEED RATE  =  3.0
;LASER INTENSITY  =  4.0
LIN {E6POS: X 1311.557, Y 58.920, Z 523.491, A 90.059, B 49.140, C -89.923, E1 0.000, E2 0.0, E3 0.0, E4 0.0, E5 0.0, E6 0.0} C_DIS
;POWDER FEED RATE  =  3.0
;LASER INTENSITY  =  4.0
LIN {E6POS: X 1306.975, Y 69.080, Z 532.509, A 86.365, B 48.301, C -94.863, E1 0.000, E2 0.0, E3 0.0, E4 0.0, E5 0.0, E6 0.0} C_DIS
;POWDER FEED RATE  =  3.0
;LASER INTENSITY  =  4.0
LIN {E6POS: X 1302.628, Y 79.240, Z 540.175, A 80.662, B 56.718, C -101.128, E1 0.000, E2 0.0, E3 0.0, E4 0.0, E5 0.0, E6 0.0} C_DIS
;POWDER FEED RATE  =  3.0
;LASER INTENSITY  =  4.0
LIN {E6POS: X 1297.559, Y 89.400, Z 544.459, A 67.919, B 69.831, C -113.373, E1 0.000, E2 0.0, E3 0.0, E4 0.0, E5 0.0, E6 0.0} C_DIS
;POWDER FEED RATE  =  3.0
;LASER INTENSITY  =  4.0
LIN {E6POS: X 1291.837, Y 99.560, Z 546.037, A 45.390, B 77.542, C -135.292, E1 0.000, E2 0.0, E3 0.0, E4 0.0, E5 0.0, E6 0.0} C_DIS
;POWDER FEED RATE  =  3.0
;LASER INTENSITY  =  4.0
LIN {E6POS: X 1285.788, Y 109.720, Z 546.262, A 30.994, B 79.093, C -149.465, E1 0.000, E2 0.0, E3 0.0, E4 0.0, E5 0.0, E6 0.0} C_DIS
;POWDER FEED RATE  =  3.0
;LASER INTENSITY  =  4.0
LIN {E6POS: X 1279.685, Y 119.880, Z 546.262, A 30.994, B 78.472, C -149.519, E1 0.000, E2 0.0, E3 0.0, E4 0.0, E5 0.0, E6 0.0} C_DIS
;POWDER FEED RATE  =  3.0
;LASER INTENSITY  =  4.0
LIN {E6POS: X 1273.581, Y 130.040, Z 546.262, A 30.994, B 77.778, C -149.583, E1 0.000, E2 0.0, E3 0.0, E4 0.0, E5 0.0, E6 0.0} C_DIS
;POWDER FEED RATE  =  3.0
;LASER INTENSITY  =  4.0
LIN {E6POS: X 1267.478, Y 140.200, Z 546.262, A 30.994, B 76.996, C -149.659, E1 0.000, E2 0.0, E3 0.0, E4 0.0, E5 0.0, E6 0.0} C_DIS
;POWDER FEED RATE  =  3.0
;LASER INTENSITY  =  4.0
>>>>>>>>>>>>>>>>>>>>>>>>>>>>POWDER FEED OFF  at=START
>>>>>>>>>>>>>>>>>>>>>>>>>>>>LASER OFF at=START
>>>>>>>>>>>>>>>>>>>>>>>>>>>>GAS SUPPLY OFF  at=START
LIN {E6POS: X 1267.478, Y 140.200, Z 546.262, A 30.994, B 76.996, C -149.659, E1 0.000, E2 0.0, E3 0.0, E4 0.0, E5 0.0, E6 0.0} C_DIS
LIN {E6POS: X 1273.581, Y 130.040, Z 546.262, A 30.994, B 77.778, C -149.583, E1 0.000, E2 0.0, E3 0.0, E4 0.0, E5 0.0, E6 0.0} C_DIS
LIN {E6POS: X 1273.581, Y 130.040, Z 546.262, A 30.994, B 77.778, C -149.583, E1 0.000, E2 0.0, E3 0.0, E4 0.0, E5 0.0, E6 0.0} C_DIS
>>>>>>>>>>>>>>>>>>>>>>>>>>>>GAS SUPPLY ON at=END
>>>>>>>>>>>>>>>>>>>>>>>>>>>>POWDER FEED ON at=END
>>>>>>>>>>>>>>>>>>>>>>>>>>>>LASER ON at=END
LIN {E6POS: X 1376.484, Y -12.200, Z 508.929, A -147.004, B 85.717, C 32.923, E1 0.000, E2 0.0, E3 0.0, E4 0.0, E5 0.0, E6 0.0} C_DIS
;POWDER FEED RATE  =  3.0
;LASER INTENSITY  =  4.0
LIN {E6POS: X 1369.806, Y -2.040, Z 508.929, A -146.053, B 85.475, C 33.864, E1 0.000, E2 0.0, E3 0.0, E4 0.0, E5 0.0, E6 0.0} C_DIS
;POWDER FEED RATE  =  3.0
;LASER INTENSITY  =  4.0
LIN {E6POS: X 1362.644, Y 8.120, Z 508.929, A -143.323, B 85.137, C 36.578, E1 0.000, E2 0.0, E3 0.0, E4 0.0, E5 0.0, E6 0.0} C_DIS
;POWDER FEED RATE  =  3.0
;LASER INTENSITY  =  4.0
LIN {E6POS: X 1354.511, Y 18.280, Z 508.929, A -139.171, B 84.720, C 40.709, E1 0.000, E2 0.0, E3 0.0, E4 0.0, E5 0.0, E6 0.0} C_DIS
;POWDER FEED RATE  =  3.0
;LASER INTENSITY  =  4.0
LIN {E6POS: X 1345.233, Y 28.440, Z 509.169, A 175.032, B 86.045, C -4.957, E1 0.000, E2 0.0, E3 0.0, E4 0.0, E5 0.0, E6 0.0} C_DIS
;POWDER FEED RATE  =  3.0
;LASER INTENSITY  =  4.0
LIN {E6POS: X 1335.865, Y 38.600, Z 510.846, A 104.267, B 76.586, C -75.349, E1 0.000, E2 0.0, E3 0.0, E4 0.0, E5 0.0, E6 0.0} C_DIS
;POWDER FEED RATE  =  3.0
;LASER INTENSITY  =  4.0
LIN {E6POS: X 1327.776, Y 48.760, Z 515.398, A 93.059, B 58.411, C -86.411, E1 0.000, E2 0.0, E3 0.0, E4 0.0, E5 0.0, E6 0.0} C_DIS
;POWDER FEED RATE  =  3.0
;LASER INTENSITY  =  4.0
LIN {E6POS: X 1321.889, Y 58.920, Z 523.543, A 89.287, B 47.221, C -90.972, E1 0.000, E2 0.0, E3 0.0, E4 0.0, E5 0.0, E6 0.0} C_DIS
;POWDER FEED RATE  =  3.0
;LASER INTENSITY  =  4.0
LIN {E6POS: X 1317.368, Y 69.080, Z 533.126, A 86.229, B 46.534, C -95.189, E1 0.000, E2 0.0, E3 0.0, E4 0.0, E5 0.0, E6 0.0} C_DIS
;POWDER FEED RATE  =  3.0
;LASER INTENSITY  =  4.0
LIN {E6POS: X 1312.936, Y 79.240, Z 541.271, A 81.221, B 55.199, C -100.651, E1 0.000, E2 0.0, E3 0.0, E4 0.0, E5 0.0, E6 0.0} C_DIS
;POWDER FEED RATE  =  3.0
;LASER INTENSITY  =  4.0
LIN {E6POS: X 1307.594, Y 89.400, Z 545.823, A 69.607, B 69.029, C -111.709, E1 0.000, E2 0.0, E3 0.0, E4 0.0, E5 0.0, E6 0.0} C_DIS
;POWDER FEED RATE  =  3.0
;LASER INTENSITY  =  4.0
LIN {E6POS: X 1301.459, Y 99.560, Z 547.500, A 47.878, B 77.509, C -132.805, E1 0.000, E2 0.0, E3 0.0, E4 0.0, E5 0.0, E6 0.0} C_DIS
;POWDER FEED RATE  =  3.0
;LASER INTENSITY  =  4.0
LIN {E6POS: X 1294.929, Y 109.720, Z 547.740, A 32.996, B 79.355, C -147.457, E1 0.000, E2 0.0, E3 0.0, E4 0.0, E5 0.0, E6 0.0} C_DIS
;POWDER FEED RATE  =  3.0
;LASER INTENSITY  =  4.0
LIN {E6POS: X 1288.332, Y 119.880, Z 547.740, A 32.996, B 78.778, C -147.508, E1 0.000, E2 0.0, E3 0.0, E4 0.0, E5 0.0, E6 0.0} C_DIS
;POWDER FEED RATE  =  3.0
;LASER INTENSITY  =  4.0
LIN {E6POS: X 1281.735, Y 130.040, Z 547.740, A 32.996, B 78.135, C -147.567, E1 0.000, E2 0.0, E3 0.0, E4 0.0, E5 0.0, E6 0.0} C_DIS
;POWDER FEED RATE  =  3.0
;LASER INTENSITY  =  4.0
LIN {E6POS: X 1275.138, Y 140.200, Z 547.740, A 32.996, B 77.415, C -147.637, E1 0.000, E2 0.0, E3 0.0, E4 0.0, E5 0.0, E6 0.0} C_DIS
;POWDER FEED RATE  =  3.0
;LASER INTENSITY  =  4.0
>>>>>>>>>>>>>>>>>>>>>>>>>>>>POWDER FEED OFF  at=START
>>>>>>>>>>>>>>>>>>>>>>>>>>>>LASER OFF at=START
>>>>>>>>>>>>>>>>>>>>>>>>>>>>GAS SUPPLY OFF  at=START
LIN {E6POS: X 1275.138, Y 140.200, Z 547.740, A 32.996, B 77.415, C -147.637, E1 0.000, E2 0.0, E3 0.0, E4 0.0, E5 0.0, E6 0.0} C_DIS
LIN {E6POS: X 1281.735, Y 130.040, Z 547.740, A 32.996, B 78.135, C -147.567, E1 0.000, E2 0.0, E3 0.0, E4 0.0, E5 0.0, E6 0.0} C_DIS
LIN {E6POS: X 1281.735, Y 130.040, Z 547.740, A 32.996, B 78.135, C -147.567, E1 0.000, E2 0.0, E3 0.0, E4 0.0, E5 0.0, E6 0.0} C_DIS
>>>>>>>>>>>>>>>>>>>>>>>>>>>>GAS SUPPLY ON at=END
>>>>>>>>>>>>>>>>>>>>>>>>>>>>POWDER FEED ON at=END
>>>>>>>>>>>>>>>>>>>>>>>>>>>>LASER ON at=END
LIN {E6POS: X 1386.881, Y -12.200, Z 508.399, A -145.223, B 87.366, C 34.749, E1 0.000, E2 0.0, E3 0.0, E4 0.0, E5 0.0, E6 0.0} C_DIS
;POWDER FEED RATE  =  3.0
;LASER INTENSITY  =  4.0
LIN {E6POS: X 1379.757, Y -2.040, Z 508.399, A -144.445, B 87.222, C 35.523, E1 0.000, E2 0.0, E3 0.0, E4 0.0, E5 0.0, E6 0.0} C_DIS
;POWDER FEED RATE  =  3.0
;LASER INTENSITY  =  4.0
LIN {E6POS: X 1372.219, Y 8.120, Z 508.399, A -142.198, B 87.029, C 37.765, E1 0.000, E2 0.0, E3 0.0, E4 0.0, E5 0.0, E6 0.0} C_DIS
;POWDER FEED RATE  =  3.0
;LASER INTENSITY  =  4.0
LIN {E6POS: X 1363.856, Y 18.280, Z 508.399, A -138.737, B 86.801, C 41.219, E1 0.000, E2 0.0, E3 0.0, E4 0.0, E5 0.0, E6 0.0} C_DIS
;POWDER FEED RATE  =  3.0
;LASER INTENSITY  =  4.0
LIN {E6POS: X 1354.539, Y 28.440, Z 508.650, A 138.843, B 86.882, C -41.115, E1 0.000, E2 0.0, E3 0.0, E4 0.0, E5 0.0, E6 0.0} C_DIS
;POWDER FEED RATE  =  3.0
;LASER INTENSITY  =  4.0
LIN {E6POS: X 1345.285, Y 38.600, Z 510.409, A 96.885, B 74.853, C -82.870, E1 0.000, E2 0.0, E3 0.0, E4 0.0, E5 0.0, E6 0.0} C_DIS
;POWDER FEED RATE  =  3.0
;LASER INTENSITY  =  4.0
LIN {E6POS: X 1337.394, Y 48.760, Z 515.184, A 90.901, B 56.535, C -88.919, E1 0.000, E2 0.0, E3 0.0, E4 0.0, E5 0.0, E6 0.0} C_DIS
;POWDER FEED RATE  =  3.0
;LASER INTENSITY  =  4.0
LIN {E6POS: X 1331.724, Y 58.920, Z 523.729, A 88.419, B 45.644, C -92.210, E1 0.000, E2 0.0, E3 0.0, E4 0.0, E5 0.0, E6 0.0} C_DIS
;POWDER FEED RATE  =  3.0
;LASER INTENSITY  =  4.0
LIN {E6POS: X 1327.356, Y 69.080, Z 533.781, A 86.017, B 45.130, C -95.611, E1 0.000, E2 0.0, E3 0.0, E4 0.0, E5 0.0, E6 0.0} C_DIS
;POWDER FEED RATE  =  3.0
;LASER INTENSITY  =  4.0
LIN {E6POS: X 1322.925, Y 79.240, Z 542.326, A 81.691, B 54.010, C -100.231, E1 0.000, E2 0.0, E3 0.0, E4 0.0, E5 0.0, E6 0.0} C_DIS
;POWDER FEED RATE  =  3.0
;LASER INTENSITY  =  4.0
LIN {E6POS: X 1317.375, Y 89.400, Z 547.101, A 71.161, B 68.471, C -110.142, E1 0.000, E2 0.0, E3 0.0, E4 0.0, E5 0.0, E6 0.0} C_DIS
;POWDER FEED RATE  =  3.0
;LASER INTENSITY  =  4.0
LIN {E6POS: X 1310.874, Y 99.560, Z 548.860, A 50.228, B 77.664, C -130.431, E1 0.000, E2 0.0, E3 0.0, E4 0.0, E5 0.0, E6 0.0} C_DIS
;POWDER FEED RATE  =  3.0
;LASER INTENSITY  =  4.0
LIN {E6POS: X 1303.898, Y 109.720, Z 549.111, A 34.777, B 79.801, C -145.649, E1 0.000, E2 0.0, E3 0.0, E4 0.0, E5 0.0, E6 0.0} C_DIS
;POWDER FEED RATE  =  3.0
;LASER INTENSITY  =  4.0
LIN {E6POS: X 1296.843, Y 119.880, Z 549.111, A 34.777, B 79.283, C -145.694, E1 0.000, E2 0.0, E3 0.0, E4 0.0, E5 0.0, E6 0.0} C_DIS
;POWDER FEED RATE  =  3.0
;LASER INTENSITY  =  4.0
LIN {E6POS: X 1289.787, Y 130.040, Z 549.111, A 34.777, B 78.711, C -145.746, E1 0.000, E2 0.0, E3 0.0, E4 0.0, E5 0.0, E6 0.0} C_DIS
;POWDER FEED RATE  =  3.0
;LASER INTENSITY  =  4.0
LIN {E6POS: X 1282.732, Y 140.200, Z 549.111, A 34.777, B 78.075, C -145.806, E1 0.000, E2 0.0, E3 0.0, E4 0.0, E5 0.0, E6 0.0} C_DIS
;POWDER FEED RATE  =  3.0
;LASER INTENSITY  =  4.0
>>>>>>>>>>>>>>>>>>>>>>>>>>>>POWDER FEED OFF  at=START
>>>>>>>>>>>>>>>>>>>>>>>>>>>>LASER OFF at=START
>>>>>>>>>>>>>>>>>>>>>>>>>>>>GAS SUPPLY OFF  at=START
LIN {E6POS: X 1282.732, Y 140.200, Z 549.111, A 34.777, B 78.075, C -145.806, E1 0.000, E2 0.0, E3 0.0, E4 0.0, E5 0.0, E6 0.0} C_DIS
LIN {E6POS: X 1289.787, Y 130.040, Z 549.111, A 34.777, B 78.711, C -145.746, E1 0.000, E2 0.0, E3 0.0, E4 0.0, E5 0.0, E6 0.0} C_DIS
LIN {E6POS: X 1289.787, Y 130.040, Z 549.111, A 34.777, B 78.711, C -145.746, E1 0.000, E2 0.0, E3 0.0, E4 0.0, E5 0.0, E6 0.0} C_DIS
>>>>>>>>>>>>>>>>>>>>>>>>>>>>GAS SUPPLY ON at=END
>>>>>>>>>>>>>>>>>>>>>>>>>>>>POWDER FEED ON at=END
>>>>>>>>>>>>>>>>>>>>>>>>>>>>LASER ON at=END
LIN {E6POS: X 1396.468, Y -12.200, Z 508.184, A -143.673, B 89.612, C 36.326, E1 0.000, E2 0.0, E3 0.0, E4 0.0, E5 0.0, E6 0.0} C_DIS
;POWDER FEED RATE  =  3.0
;LASER INTENSITY  =  4.0
LIN {E6POS: X 1388.939, Y -2.040, Z 508.184, A -143.042, B 89.592, C 36.958, E1 0.000, E2 0.0, E3 0.0, E4 0.0, E5 0.0, E6 0.0} C_DIS
;POWDER FEED RATE  =  3.0
;LASER INTENSITY  =  4.0
LIN {E6POS: X 1381.062, Y 8.120, Z 508.184, A -141.208, B 89.566, C 38.791, E1 0.000, E2 0.0, E3 0.0, E4 0.0, E5 0.0, E6 0.0} C_DIS
;POWDER FEED RATE  =  3.0
;LASER INTENSITY  =  4.0
LIN {E6POS: X 1372.490, Y 18.280, Z 508.184, A -138.349, B 89.536, C 41.650, E1 0.000, E2 0.0, E3 0.0, E4 0.0, E5 0.0, E6 0.0} C_DIS
;POWDER FEED RATE  =  3.0
;LASER INTENSITY  =  4.0
LIN {E6POS: X 1363.141, Y 28.440, Z 508.445, A 94.088, B 85.867, C -85.901, E1 0.000, E2 0.0, E3 0.0, E4 0.0, E5 0.0, E6 0.0} C_DIS
;POWDER FEED RATE  =  3.0
;LASER INTENSITY  =  4.0
LIN {E6POS: X 1354.009, Y 38.600, Z 510.267, A 89.768, B 72.855, C -90.242, E1 0.000, E2 0.0, E3 0.0, E4 0.0, E5 0.0, E6 0.0} C_DIS
;POWDER FEED RATE  =  3.0
;LASER INTENSITY  =  4.0
LIN {E6POS: X 1346.353, Y 48.760, Z 515.213, A 88.545, B 54.877, C -91.779, E1 0.000, E2 0.0, E3 0.0, E4 0.0, E5 0.0, E6 0.0} C_DIS
;POWDER FEED RATE  =  3.0
;LASER INTENSITY  =  4.0
LIN {E6POS: X 1340.977, Y 58.920, Z 524.063, A 87.423, B 44.417, C -93.679, E1 0.000, E2 0.0, E3 0.0, E4 0.0, E5 0.0, E6 0.0} C_DIS
;POWDER FEED RATE  =  3.0
;LASER INTENSITY  =  4.0
LIN {E6POS: X 1336.862, Y 69.080, Z 534.475, A 85.722, B 44.091, C -96.137, E1 0.000, E2 0.0, E3 0.0, E4 0.0, E5 0.0, E6 0.0} C_DIS
;POWDER FEED RATE  =  3.0
;LASER INTENSITY  =  4.0
LIN {E6POS: X 1332.531, Y 79.240, Z 543.326, A 82.089, B 53.170, C -99.849, E1 0.000, E2 0.0, E3 0.0, E4 0.0, E5 0.0, E6 0.0} C_DIS
;POWDER FEED RATE  =  3.0
;LASER INTENSITY  =  4.0
LIN {E6POS: X 1326.847, Y 89.400, Z 548.271, A 72.626, B 68.182, C -108.626, E1 0.000, E2 0.0, E3 0.0, E4 0.0, E5 0.0, E6 0.0} C_DIS
;POWDER FEED RATE  =  3.0
;LASER INTENSITY  =  4.0
LIN {E6POS: X 1320.034, Y 99.560, Z 550.094, A 52.488, B 78.026, C -128.122, E1 0.000, E2 0.0, E3 0.0, E4 0.0, E5 0.0, E6 0.0} C_DIS
;POWDER FEED RATE  =  3.0
;LASER INTENSITY  =  4.0
LIN {E6POS: X 1312.658, Y 109.720, Z 550.354, A 36.327, B 80.443, C -144.055, E1 0.000, E2 0.0, E3 0.0, E4 0.0, E5 0.0, E6 0.0} C_DIS
;POWDER FEED RATE  =  3.0
;LASER INTENSITY  =  4.0
LIN {E6POS: X 1305.187, Y 119.880, Z 550.354, A 36.327, B 79.998, C -144.091, E1 0.000, E2 0.0, E3 0.0, E4 0.0, E5 0.0, E6 0.0} C_DIS
;POWDER FEED RATE  =  3.0
;LASER INTENSITY  =  4.0
LIN {E6POS: X 1297.717, Y 130.040, Z 550.354, A 36.327, B 79.511, C -144.133, E1 0.000, E2 0.0, E3 0.0, E4 0.0, E5 0.0, E6 0.0} C_DIS
;POWDER FEED RATE  =  3.0
;LASER INTENSITY  =  4.0
LIN {E6POS: X 1290.246, Y 140.200, Z 550.354, A 36.327, B 78.973, C -144.181, E1 0.000, E2 0.0, E3 0.0, E4 0.0, E5 0.0, E6 0.0} C_DIS
;POWDER FEED RATE  =  3.0
;LASER INTENSITY  =  4.0
>>>>>>>>>>>>>>>>>>>>>>>>>>>>POWDER FEED OFF  at=START
>>>>>>>>>>>>>>>>>>>>>>>>>>>>LASER OFF at=START
>>>>>>>>>>>>>>>>>>>>>>>>>>>>GAS SUPPLY OFF  at=START
LIN {E6POS: X 1290.246, Y 140.200, Z 550.354, A 36.327, B 78.973, C -144.181, E1 0.000, E2 0.0, E3 0.0, E4 0.0, E5 0.0, E6 0.0} C_DIS
LIN {E6POS: X 1297.717, Y 130.040, Z 550.354, A 36.327, B 79.511, C -144.133, E1 0.000, E2 0.0, E3 0.0, E4 0.0, E5 0.0, E6 0.0} C_DIS
LIN {E6POS: X 1297.717, Y 130.040, Z 550.354, A 36.327, B 79.511, C -144.133, E1 0.000, E2 0.0, E3 0.0, E4 0.0, E5 0.0, E6 0.0} C_DIS
>>>>>>>>>>>>>>>>>>>>>>>>>>>>GAS SUPPLY ON at=END
>>>>>>>>>>>>>>>>>>>>>>>>>>>>POWDER FEED ON at=END
>>>>>>>>>>>>>>>>>>>>>>>>>>>>LASER ON at=END
LIN {E6POS: X 1405.225, Y -12.200, Z 508.288, A 37.655, B 87.832, C -142.364, E1 0.000, E2 0.0, E3 0.0, E4 0.0, E5 0.0, E6 0.0} C_DIS
;POWDER FEED RATE  =  3.0
;LASER INTENSITY  =  4.0
LIN {E6POS: X 1397.337, Y -2.040, Z 508.288, A 38.165, B 87.725, C -141.857, E1 0.000, E2 0.0, E3 0.0, E4 0.0, E5 0.0, E6 0.0} C_DIS
;POWDER FEED RATE  =  3.0
;LASER INTENSITY  =  4.0
LIN {E6POS: X 1389.159, Y 8.120, Z 508.288, A 39.651, B 87.592, C -140.374, E1 0.000, E2 0.0, E3 0.0, E4 0.0, E5 0.0, E6 0.0} C_DIS
;POWDER FEED RATE  =  3.0
;LASER INTENSITY  =  4.0
LIN {E6POS: X 1380.400, Y 18.280, Z 508.288, A 41.992, B 87.448, C -138.036, E1 0.000, E2 0.0, E3 0.0, E4 0.0, E5 0.0, E6 0.0} C_DIS
;POWDER FEED RATE  =  3.0
;LASER INTENSITY  =  4.0
LIN {E6POS: X 1371.026, Y 28.440, Z 508.554, A 72.890, B 83.435, C -107.216, E1 0.000, E2 0.0, E3 0.0, E4 0.0, E5 0.0, E6 0.0} C_DIS
;POWDER FEED RATE  =  3.0
;LASER INTENSITY  =  4.0
LIN {E6POS: X 1362.025, Y 38.600, Z 510.420, A 83.780, B 70.814, C -96.582, E1 0.000, E2 0.0, E3 0.0, E4 0.0, E5 0.0, E6 0.0} C_DIS
;POWDER FEED RATE  =  3.0
;LASER INTENSITY  =  4.0
LIN {E6POS: X 1354.638, Y 48.760, Z 515.483, A 86.279, B 53.541, C -94.623, E1 0.000, E2 0.0, E3 0.0, E4 0.0, E5 0.0, E6 0.0} C_DIS
;POWDER FEED RATE  =  3.0
;LASER INTENSITY  =  4.0
LIN {E6POS: X 1349.633, Y 58.920, Z 524.544, A 86.434, B 43.563, C -95.167, E1 0.000, E2 0.0, E3 0.0, E4 0.0, E5 0.0, E6 0.0} C_DIS
;POWDER FEED RATE  =  3.0
;LASER INTENSITY  =  4.0
LIN {E6POS: X 1345.869, Y 69.080, Z 535.203, A 85.408, B 43.413, C -96.666, E1 0.000, E2 0.0, E3 0.0, E4 0.0, E5 0.0, E6 0.0} C_DIS
;POWDER FEED RATE  =  3.0
;LASER INTENSITY  =  4.0
LIN {E6POS: X 1341.734, Y 79.240, Z 544.264, A 82.415, B 52.655, C -99.509, E1 0.000, E2 0.0, E3 0.0, E4 0.0, E5 0.0, E6 0.0} C_DIS
;POWDER FEED RATE  =  3.0
;LASER INTENSITY  =  4.0
LIN {E6POS: X 1335.992, Y 89.400, Z 549.327, A 73.924, B 68.109, C -107.253, E1 0.000, E2 0.0, E3 0.0, E4 0.0, E5 0.0, E6 0.0} C_DIS
;POWDER FEED RATE  =  3.0
;LASER INTENSITY  =  4.0
LIN {E6POS: X 1328.924, Y 99.560, Z 551.193, A 54.571, B 78.490, C -125.981, E1 0.000, E2 0.0, E3 0.0, E4 0.0, E5 0.0, E6 0.0} C_DIS
;POWDER FEED RATE  =  3.0
;LASER INTENSITY  =  4.0
LIN {E6POS: X 1321.195, Y 109.720, Z 551.459, A 37.655, B 81.151, C -142.676, E1 0.000, E2 0.0, E3 0.0, E4 0.0, E5 0.0, E6 0.0} C_DIS
;POWDER FEED RATE  =  3.0
;LASER INTENSITY  =  4.0
LIN {E6POS: X 1313.355, Y 119.880, Z 551.459, A 37.655, B 80.777, C -142.705, E1 0.000, E2 0.0, E3 0.0, E4 0.0, E5 0.0, E6 0.0} C_DIS
;POWDER FEED RATE  =  3.0
;LASER INTENSITY  =  4.0
LIN {E6POS: X 1305.515, Y 130.040, Z 551.459, A 37.655, B 80.371, C -142.737, E1 0.000, E2 0.0, E3 0.0, E4 0.0, E5 0.0, E6 0.0} C_DIS
;POWDER FEED RATE  =  3.0
;LASER INTENSITY  =  4.0
LIN {E6POS: X 1297.675, Y 140.200, Z 551.459, A 37.655, B 79.928, C -142.774, E1 0.000, E2 0.0, E3 0.0, E4 0.0, E5 0.0, E6 0.0} C_DIS
;POWDER FEED RATE  =  3.0
;LASER INTENSITY  =  4.0
>>>>>>>>>>>>>>>>>>>>>>>>>>>>POWDER FEED OFF  at=START
>>>>>>>>>>>>>>>>>>>>>>>>>>>>LASER OFF at=START
>>>>>>>>>>>>>>>>>>>>>>>>>>>>GAS SUPPLY OFF  at=START
LIN {E6POS: X 1297.675, Y 140.200, Z 551.459, A 37.655, B 79.928, C -142.774, E1 0.000, E2 0.0, E3 0.0, E4 0.0, E5 0.0, E6 0.0} C_DIS
LIN {E6POS: X 1305.515, Y 130.040, Z 551.459, A 37.655, B 80.371, C -142.737, E1 0.000, E2 0.0, E3 0.0, E4 0.0, E5 0.0, E6 0.0} C_DIS
LIN {E6POS: X 1305.515, Y 130.040, Z 551.459, A 37.655, B 80.371, C -142.737, E1 0.000, E2 0.0, E3 0.0, E4 0.0, E5 0.0, E6 0.0} C_DIS
>>>>>>>>>>>>>>>>>>>>>>>>>>>>GAS SUPPLY ON at=END
>>>>>>>>>>>>>>>>>>>>>>>>>>>>POWDER FEED ON at=END
>>>>>>>>>>>>>>>>>>>>>>>>>>>>LASER ON at=END
LIN {E6POS: X 1413.232, Y -12.200, Z 508.673, A 38.790, B 85.075, C -141.314, E1 0.000, E2 0.0, E3 0.0, E4 0.0, E5 0.0, E6 0.0} C_DIS
;POWDER FEED RATE  =  3.0
;LASER INTENSITY  =  4.0
LIN {E6POS: X 1405.026, Y -2.040, Z 508.673, A 39.197, B 84.848, C -140.917, E1 0.000, E2 0.0, E3 0.0, E4 0.0, E5 0.0, E6 0.0} C_DIS
;POWDER FEED RATE  =  3.0
;LASER INTENSITY  =  4.0
LIN {E6POS: X 1396.581, Y 8.120, Z 508.673, A 40.391, B 84.575, C -139.736, E1 0.000, E2 0.0, E3 0.0, E4 0.0, E5 0.0, E6 0.0} C_DIS
;POWDER FEED RATE  =  3.0
;LASER INTENSITY  =  4.0
LIN {E6POS: X 1387.658, Y 18.280, Z 508.673, A 42.290, B 84.293, C -137.852, E1 0.000, E2 0.0, E3 0.0, E4 0.0, E5 0.0, E6 0.0} C_DIS
;POWDER FEED RATE  =  3.0
;LASER INTENSITY  =  4.0
LIN {E6POS: X 1378.266, Y 28.440, Z 508.944, A 63.323, B 80.585, C -116.990, E1 0.000, E2 0.0, E3 0.0, E4 0.0, E5 0.0, E6 0.0} C_DIS
;POWDER FEED RATE  =  3.0
;LASER INTENSITY  =  4.0
LIN {E6POS: X 1369.402, Y 38.600, Z 510.835, A 78.770, B 68.833, C -102.019, E1 0.000, E2 0.0, E3 0.0, E4 0.0, E5 0.0, E6 0.0} C_DIS
;POWDER FEED RATE  =  3.0
;LASER INTENSITY  =  4.0
LIN {E6POS: X 1362.313, Y 48.760, Z 515.967, A 84.118, B 52.525, C -97.397, E1 0.000, E2 0.0, E3 0.0, E4 0.0, E5 0.0, E6 0.0} C_DIS
;POWDER FEED RATE  =  3.0
;LASER INTENSITY  =  4.0
LIN {E6POS: X 1357.742, Y 58.920, Z 525.151, A 85.468, B 43.045, C -96.623, E1 0.000, E2 0.0, E3 0.0, E4 0.0, E5 0.0, E6 0.0} C_DIS
;POWDER FEED RATE  =  3.0
;LASER INTENSITY  =  4.0
LIN {E6POS: X 1354.417, Y 69.080, Z 535.957, A 85.093, B 43.049, C -97.169, E1 0.000, E2 0.0, E3 0.0, E4 0.0, E5 0.0, E6 0.0} C_DIS
;POWDER FEED RATE  =  3.0
;LASER INTENSITY  =  4.0
LIN {E6POS: X 1350.563, Y 79.240, Z 545.141, A 82.693, B 52.422, C -99.191, E1 0.000, E2 0.0, E3 0.0, E4 0.0, E5 0.0, E6 0.0} C_DIS
;POWDER FEED RATE  =  3.0
;LASER INTENSITY  =  4.0
LIN {E6POS: X 1344.829, Y 89.400, Z 550.273, A 75.091, B 68.219, C -105.998, E1 0.000, E2 0.0, E3 0.0, E4 0.0, E5 0.0, E6 0.0} C_DIS
;POWDER FEED RATE  =  3.0
;LASER INTENSITY  =  4.0
LIN {E6POS: X 1337.559, Y 99.560, Z 552.164, A 56.511, B 79.027, C -123.977, E1 0.000, E2 0.0, E3 0.0, E4 0.0, E5 0.0, E6 0.0} C_DIS
;POWDER FEED RATE  =  3.0
;LASER INTENSITY  =  4.0
LIN {E6POS: X 1329.521, Y 109.720, Z 552.434, A 38.790, B 81.894, C -141.491, E1 0.000, E2 0.0, E3 0.0, E4 0.0, E5 0.0, E6 0.0} C_DIS
;POWDER FEED RATE  =  3.0
;LASER INTENSITY  =  4.0
LIN {E6POS: X 1321.355, Y 119.880, Z 552.434, A 38.790, B 81.586, C -141.513, E1 0.000, E2 0.0, E3 0.0, E4 0.0, E5 0.0, E6 0.0} C_DIS
;POWDER FEED RATE  =  3.0
;LASER INTENSITY  =  4.0
LIN {E6POS: X 1313.189, Y 130.040, Z 552.434, A 38.790, B 81.254, C -141.537, E1 0.000, E2 0.0, E3 0.0, E4 0.0, E5 0.0, E6 0.0} C_DIS
;POWDER FEED RATE  =  3.0
;LASER INTENSITY  =  4.0
LIN {E6POS: X 1305.023, Y 140.200, Z 552.434, A 38.790, B 80.895, C -141.564, E1 0.000, E2 0.0, E3 0.0, E4 0.0, E5 0.0, E6 0.0} C_DIS
;POWDER FEED RATE  =  3.0
;LASER INTENSITY  =  4.0
>>>>>>>>>>>>>>>>>>>>>>>>>>>>POWDER FEED OFF  at=START
>>>>>>>>>>>>>>>>>>>>>>>>>>>>LASER OFF at=START
>>>>>>>>>>>>>>>>>>>>>>>>>>>>GAS SUPPLY OFF  at=START
LIN {E6POS: X 1305.023, Y 140.200, Z 552.434, A 38.790, B 80.895, C -141.564, E1 0.000, E2 0.0, E3 0.0, E4 0.0, E5 0.0, E6 0.0} C_DIS
LIN {E6POS: X 1313.189, Y 130.040, Z 552.434, A 38.790, B 81.254, C -141.537, E1 0.000, E2 0.0, E3 0.0, E4 0.0, E5 0.0, E6 0.0} C_DIS
LIN {E6POS: X 1313.189, Y 130.040, Z 552.434, A 38.790, B 81.254, C -141.537, E1 0.000, E2 0.0, E3 0.0, E4 0.0, E5 0.0, E6 0.0} C_DIS
>>>>>>>>>>>>>>>>>>>>>>>>>>>>GAS SUPPLY ON at=END
>>>>>>>>>>>>>>>>>>>>>>>>>>>>POWDER FEED ON at=END
>>>>>>>>>>>>>>>>>>>>>>>>>>>>LASER ON at=END
LIN {E6POS: X 1420.567, Y -12.200, Z 509.304, A 39.754, B 82.195, C -140.508, E1 0.000, E2 0.0, E3 0.0, E4 0.0, E5 0.0, E6 0.0} C_DIS
;POWDER FEED RATE  =  3.0
;LASER INTENSITY  =  4.0
LIN {E6POS: X 1412.084, Y -2.040, Z 509.304, A 40.076, B 81.862, C -140.209, E1 0.000, E2 0.0, E3 0.0, E4 0.0, E5 0.0, E6 0.0} C_DIS
;POWDER FEED RATE  =  3.0
;LASER INTENSITY  =  4.0
LIN {E6POS: X 1403.406, Y 8.120, Z 509.304, A 41.025, B 81.478, C -139.289, E1 0.000, E2 0.0, E3 0.0, E4 0.0, E5 0.0, E6 0.0} C_DIS
;POWDER FEED RATE  =  3.0
;LASER INTENSITY  =  4.0
LIN {E6POS: X 1394.339, Y 18.280, Z 509.304, A 42.549, B 81.097, C -137.797, E1 0.000, E2 0.0, E3 0.0, E4 0.0, E5 0.0, E6 0.0} C_DIS
;POWDER FEED RATE  =  3.0
;LASER INTENSITY  =  4.0
LIN {E6POS: X 1384.933, Y 28.440, Z 509.576, A 58.092, B 77.658, C -122.512, E1 0.000, E2 0.0, E3 0.0, E4 0.0, E5 0.0, E6 0.0} C_DIS
;POWDER FEED RATE  =  3.0
;LASER INTENSITY  =  4.0
LIN {E6POS: X 1376.212, Y 38.600, Z 511.476, A 74.514, B 66.977, C -106.753, E1 0.000, E2 0.0, E3 0.0, E4 0.0, E5 0.0, E6 0.0} C_DIS
;POWDER FEED RATE  =  3.0
;LASER INTENSITY  =  4.0
LIN {E6POS: X 1369.444, Y 48.760, Z 516.635, A 82.040, B 51.809, C -100.088, E1 0.000, E2 0.0, E3 0.0, E4 0.0, E5 0.0, E6 0.0} C_DIS
;POWDER FEED RATE  =  3.0
;LASER INTENSITY  =  4.0
LIN {E6POS: X 1365.361, Y 58.920, Z 525.866, A 84.523, B 42.830, C -98.029, E1 0.000, E2 0.0, E3 0.0, E4 0.0, E5 0.0, E6 0.0} C_DIS
;POWDER FEED RATE  =  3.0
;LASER INTENSITY  =  4.0
LIN {E6POS: X 1362.546, Y 69.080, Z 536.726, A 84.782, B 42.960, C -97.632, E1 0.000, E2 0.0, E3 0.0, E4 0.0, E5 0.0, E6 0.0} C_DIS
;POWDER FEED RATE  =  3.0
;LASER INTENSITY  =  4.0
LIN {E6POS: X 1359.046, Y 79.240, Z 545.957, A 82.942, B 52.434, C -98.878, E1 0.000, E2 0.0, E3 0.0, E4 0.0, E5 0.0, E6 0.0} C_DIS
;POWDER FEED RATE  =  3.0
;LASER INTENSITY  =  4.0
LIN {E6POS: X 1353.379, Y 89.400, Z 551.116, A 76.171, B 68.488, C -104.820, E1 0.000, E2 0.0, E3 0.0, E4 0.0, E5 0.0, E6 0.0} C_DIS
;POWDER FEED RATE  =  3.0
;LASER INTENSITY  =  4.0
LIN {E6POS: X 1345.954, Y 99.560, Z 553.016, A 58.369, B 79.625, C -122.054, E1 0.000, E2 0.0, E3 0.0, E4 0.0, E5 0.0, E6 0.0} C_DIS
;POWDER FEED RATE  =  3.0
;LASER INTENSITY  =  4.0
LIN {E6POS: X 1337.649, Y 109.720, Z 553.288, A 39.754, B 82.662, C -140.478, E1 0.000, E2 0.0, E3 0.0, E4 0.0, E5 0.0, E6 0.0} C_DIS
;POWDER FEED RATE  =  3.0
;LASER INTENSITY  =  4.0
LIN {E6POS: X 1329.198, Y 119.880, Z 553.288, A 39.754, B 82.414, C -140.494, E1 0.000, E2 0.0, E3 0.0, E4 0.0, E5 0.0, E6 0.0} C_DIS
;POWDER FEED RATE  =  3.0
;LASER INTENSITY  =  4.0
LIN {E6POS: X 1320.747, Y 130.040, Z 553.288, A 39.754, B 82.148, C -140.511, E1 0.000, E2 0.0, E3 0.0, E4 0.0, E5 0.0, E6 0.0} C_DIS
;POWDER FEED RATE  =  3.0
;LASER INTENSITY  =  4.0
LIN {E6POS: X 1312.296, Y 140.200, Z 553.288, A 39.754, B 81.863, C -140.531, E1 0.000, E2 0.0, E3 0.0, E4 0.0, E5 0.0, E6 0.0} C_DIS
;POWDER FEED RATE  =  3.0
;LASER INTENSITY  =  4.0
>>>>>>>>>>>>>>>>>>>>>>>>>>>>POWDER FEED OFF  at=START
>>>>>>>>>>>>>>>>>>>>>>>>>>>>LASER OFF at=START
>>>>>>>>>>>>>>>>>>>>>>>>>>>>GAS SUPPLY OFF  at=START
LIN {E6POS: X 1312.296, Y 140.200, Z 553.288, A 39.754, B 81.863, C -140.531, E1 0.000, E2 0.0, E3 0.0, E4 0.0, E5 0.0, E6 0.0} C_DIS
LIN {E6POS: X 1320.747, Y 130.040, Z 553.288, A 39.754, B 82.148, C -140.511, E1 0.000, E2 0.0, E3 0.0, E4 0.0, E5 0.0, E6 0.0} C_DIS
LIN {E6POS: X 1320.747, Y 130.040, Z 553.288, A 39.754, B 82.148, C -140.511, E1 0.000, E2 0.0, E3 0.0, E4 0.0, E5 0.0, E6 0.0} C_DIS
>>>>>>>>>>>>>>>>>>>>>>>>>>>>GAS SUPPLY ON at=END
>>>>>>>>>>>>>>>>>>>>>>>>>>>>POWDER FEED ON at=END
>>>>>>>>>>>>>>>>>>>>>>>>>>>>LASER ON at=END
LIN {E6POS: X 1427.314, Y -12.200, Z 510.142, A 40.568, B 79.303, C -139.927, E1 0.000, E2 0.0, E3 0.0, E4 0.0, E5 0.0, E6 0.0} C_DIS
;POWDER FEED RATE  =  3.0
;LASER INTENSITY  =  4.0
LIN {E6POS: X 1418.589, Y -2.040, Z 510.142, A 40.821, B 78.890, C -139.715, E1 0.000, E2 0.0, E3 0.0, E4 0.0, E5 0.0, E6 0.0} C_DIS
;POWDER FEED RATE  =  3.0
;LASER INTENSITY  =  4.0
LIN {E6POS: X 1409.709, Y 8.120, Z 510.142, A 41.566, B 78.428, C -139.017, E1 0.000, E2 0.0, E3 0.0, E4 0.0, E5 0.0, E6 0.0} C_DIS
;POWDER FEED RATE  =  3.0
;LASER INTENSITY  =  4.0
LIN {E6POS: X 1400.518, Y 18.280, Z 510.142, A 42.771, B 77.990, C -137.860, E1 0.000, E2 0.0, E3 0.0, E4 0.0, E5 0.0, E6 0.0} C_DIS
;POWDER FEED RATE  =  3.0
;LASER INTENSITY  =  4.0
LIN {E6POS: X 1391.103, Y 28.440, Z 510.413, A 54.832, B 74.838, C -126.130, E1 0.000, E2 0.0, E3 0.0, E4 0.0, E5 0.0, E6 0.0} C_DIS
;POWDER FEED RATE  =  3.0
;LASER INTENSITY  =  4.0
LIN {E6POS: X 1382.528, Y 38.600, Z 512.309, A 70.880, B 65.309, C -110.885, E1 0.000, E2 0.0, E3 0.0, E4 0.0, E5 0.0, E6 0.0} C_DIS
;POWDER FEED RATE  =  3.0
;LASER INTENSITY  =  4.0
LIN {E6POS: X 1376.099, Y 48.760, Z 517.456, A 80.046, B 51.381, C -102.660, E1 0.000, E2 0.0, E3 0.0, E4 0.0, E5 0.0, E6 0.0} C_DIS
;POWDER FEED RATE  =  3.0
;LASER INTENSITY  =  4.0
LIN {E6POS: X 1372.545, Y 58.920, Z 526.667, A 83.603, B 42.888, C -99.354, E1 0.000, E2 0.0, E3 0.0, E4 0.0, E5 0.0, E6 0.0} C_DIS
;POWDER FEED RATE  =  3.0
;LASER INTENSITY  =  4.0
LIN {E6POS: X 1370.298, Y 69.080, Z 537.503, A 84.487, B 43.113, C -98.039, E1 0.000, E2 0.0, E3 0.0, E4 0.0, E5 0.0, E6 0.0} C_DIS
;POWDER FEED RATE  =  3.0
;LASER INTENSITY  =  4.0
LIN {E6POS: X 1367.212, Y 79.240, Z 546.714, A 83.179, B 52.658, C -98.556, E1 0.000, E2 0.0, E3 0.0, E4 0.0, E5 0.0, E6 0.0} C_DIS
;POWDER FEED RATE  =  3.0
;LASER INTENSITY  =  4.0
LIN {E6POS: X 1361.664, Y 89.400, Z 551.861, A 77.198, B 68.891, C -103.689, E1 0.000, E2 0.0, E3 0.0, E4 0.0, E5 0.0, E6 0.0} C_DIS
;POWDER FEED RATE  =  3.0
;LASER INTENSITY  =  4.0
LIN {E6POS: X 1354.126, Y 99.560, Z 553.757, A 60.196, B 80.271, C -120.163, E1 0.000, E2 0.0, E3 0.0, E4 0.0, E5 0.0, E6 0.0} C_DIS
;POWDER FEED RATE  =  3.0
;LASER INTENSITY  =  4.0
LIN {E6POS: X 1345.593, Y 109.720, Z 554.028, A 40.568, B 83.444, C -139.617, E1 0.000, E2 0.0, E3 0.0, E4 0.0, E5 0.0, E6 0.0} C_DIS
;POWDER FEED RATE  =  3.0
;LASER INTENSITY  =  4.0
LIN {E6POS: X 1336.895, Y 119.880, Z 554.028, A 40.568, B 83.249, C -139.629, E1 0.000, E2 0.0, E3 0.0, E4 0.0, E5 0.0, E6 0.0} C_DIS
;POWDER FEED RATE  =  3.0
;LASER INTENSITY  =  4.0
LIN {E6POS: X 1328.197, Y 130.040, Z 554.028, A 40.568, B 83.042, C -139.641, E1 0.000, E2 0.0, E3 0.0, E4 0.0, E5 0.0, E6 0.0} C_DIS
;POWDER FEED RATE  =  3.0
;LASER INTENSITY  =  4.0
LIN {E6POS: X 1319.498, Y 140.200, Z 554.028, A 40.568, B 82.821, C -139.654, E1 0.000, E2 0.0, E3 0.0, E4 0.0, E5 0.0, E6 0.0} C_DIS
;POWDER FEED RATE  =  3.0
;LASER INTENSITY  =  4.0
>>>>>>>>>>>>>>>>>>>>>>>>>>>>POWDER FEED OFF  at=START
>>>>>>>>>>>>>>>>>>>>>>>>>>>>LASER OFF at=START
>>>>>>>>>>>>>>>>>>>>>>>>>>>>GAS SUPPLY OFF  at=START
LIN {E6POS: X 1319.498, Y 140.200, Z 554.028, A 40.568, B 82.821, C -139.654, E1 0.000, E2 0.0, E3 0.0, E4 0.0, E5 0.0, E6 0.0} C_DIS
LIN {E6POS: X 1328.197, Y 130.040, Z 554.028, A 40.568, B 83.042, C -139.641, E1 0.000, E2 0.0, E3 0.0, E4 0.0, E5 0.0, E6 0.0} C_DIS
LIN {E6POS: X 1328.197, Y 130.040, Z 554.028, A 40.568, B 83.042, C -139.641, E1 0.000, E2 0.0, E3 0.0, E4 0.0, E5 0.0, E6 0.0} C_DIS
>>>>>>>>>>>>>>>>>>>>>>>>>>>>GAS SUPPLY ON at=END
>>>>>>>>>>>>>>>>>>>>>>>>>>>>POWDER FEED ON at=END
>>>>>>>>>>>>>>>>>>>>>>>>>>>>LASER ON at=END
LIN {E6POS: X 1433.552, Y -12.200, Z 511.151, A 41.251, B 76.543, C -139.538, E1 0.000, E2 0.0, E3 0.0, E4 0.0, E5 0.0, E6 0.0} C_DIS
;POWDER FEED RATE  =  3.0
;LASER INTENSITY  =  4.0
LIN {E6POS: X 1424.621, Y -2.040, Z 511.151, A 41.446, B 76.080, C -139.400, E1 0.000, E2 0.0, E3 0.0, E4 0.0, E5 0.0, E6 0.0} C_DIS
;POWDER FEED RATE  =  3.0
;LASER INTENSITY  =  4.0
LIN {E6POS: X 1415.568, Y 8.120, Z 511.151, A 42.022, B 75.580, C -138.888, E1 0.000, E2 0.0, E3 0.0, E4 0.0, E5 0.0, E6 0.0} C_DIS
;POWDER FEED RATE  =  3.0
;LASER INTENSITY  =  4.0
LIN {E6POS: X 1406.270, Y 18.280, Z 511.151, A 42.961, B 75.124, C -138.012, E1 0.000, E2 0.0, E3 0.0, E4 0.0, E5 0.0, E6 0.0} C_DIS
;POWDER FEED RATE  =  3.0
;LASER INTENSITY  =  4.0
LIN {E6POS: X 1396.851, Y 28.440, Z 511.419, A 52.634, B 72.281, C -128.718, E1 0.000, E2 0.0, E3 0.0, E4 0.0, E5 0.0, E6 0.0} C_DIS
;POWDER FEED RATE  =  3.0
;LASER INTENSITY  =  4.0
LIN {E6POS: X 1388.423, Y 38.600, Z 513.300, A 67.793, B 63.900, C -114.447, E1 0.000, E2 0.0, E3 0.0, E4 0.0, E5 0.0, E6 0.0} C_DIS
;POWDER FEED RATE  =  3.0
;LASER INTENSITY  =  4.0
LIN {E6POS: X 1382.343, Y 48.760, Z 518.403, A 78.161, B 51.233, C -105.048, E1 0.000, E2 0.0, E3 0.0, E4 0.0, E5 0.0, E6 0.0} C_DIS
;POWDER FEED RATE  =  3.0
;LASER INTENSITY  =  4.0
LIN {E6POS: X 1379.350, Y 58.920, Z 527.535, A 82.728, B 43.195, C -100.560, E1 0.000, E2 0.0, E3 0.0, E4 0.0, E5 0.0, E6 0.0} C_DIS
;POWDER FEED RATE  =  3.0
;LASER INTENSITY  =  4.0
LIN {E6POS: X 1377.715, Y 69.080, Z 538.278, A 84.219, B 43.479, C -98.370, E1 0.000, E2 0.0, E3 0.0, E4 0.0, E5 0.0, E6 0.0} C_DIS
;POWDER FEED RATE  =  3.0
;LASER INTENSITY  =  4.0
LIN {E6POS: X 1375.090, Y 79.240, Z 547.410, A 83.420, B 53.063, C -98.212, E1 0.000, E2 0.0, E3 0.0, E4 0.0, E5 0.0, E6 0.0} C_DIS
;POWDER FEED RATE  =  3.0
;LASER INTENSITY  =  4.0
LIN {E6POS: X 1369.703, Y 89.400, Z 552.514, A 78.199, B 69.407, C -102.582, E1 0.000, E2 0.0, E3 0.0, E4 0.0, E5 0.0, E6 0.0} C_DIS
;POWDER FEED RATE  =  3.0
;LASER INTENSITY  =  4.0
LIN {E6POS: X 1362.091, Y 99.560, Z 554.394, A 62.045, B 80.949, C -118.253, E1 0.000, E2 0.0, E3 0.0, E4 0.0, E5 0.0, E6 0.0} C_DIS
;POWDER FEED RATE  =  3.0
;LASER INTENSITY  =  4.0
LIN {E6POS: X 1353.366, Y 109.720, Z 554.662, A 41.251, B 84.229, C -138.893, E1 0.000, E2 0.0, E3 0.0, E4 0.0, E5 0.0, E6 0.0} C_DIS
;POWDER FEED RATE  =  3.0
;LASER INTENSITY  =  4.0
LIN {E6POS: X 1344.456, Y 119.880, Z 554.662, A 41.251, B 84.080, C -138.901, E1 0.000, E2 0.0, E3 0.0, E4 0.0, E5 0.0, E6 0.0} C_DIS
;POWDER FEED RATE  =  3.0
;LASER INTENSITY  =  4.0
LIN {E6POS: X 1335.545, Y 130.040, Z 554.662, A 41.251, B 83.923, C -138.909, E1 0.000, E2 0.0, E3 0.0, E4 0.0, E5 0.0, E6 0.0} C_DIS
;POWDER FEED RATE  =  3.0
;LASER INTENSITY  =  4.0
LIN {E6POS: X 1326.635, Y 140.200, Z 554.662, A 41.251, B 83.757, C -138.918, E1 0.000, E2 0.0, E3 0.0, E4 0.0, E5 0.0, E6 0.0} C_DIS
;POWDER FEED RATE  =  3.0
;LASER INTENSITY  =  4.0
>>>>>>>>>>>>>>>>>>>>>>>>>>>>POWDER FEED OFF  at=START
>>>>>>>>>>>>>>>>>>>>>>>>>>>>LASER OFF at=START
>>>>>>>>>>>>>>>>>>>>>>>>>>>>GAS SUPPLY OFF  at=START
LIN {E6POS: X 1326.635, Y 140.200, Z 554.662, A 41.251, B 83.757, C -138.918, E1 0.000, E2 0.0, E3 0.0, E4 0.0, E5 0.0, E6 0.0} C_DIS
LIN {E6POS: X 1335.545, Y 130.040, Z 554.662, A 41.251, B 83.923, C -138.909, E1 0.000, E2 0.0, E3 0.0, E4 0.0, E5 0.0, E6 0.0} C_DIS
LIN {E6POS: X 1335.545, Y 130.040, Z 554.662, A 41.251, B 83.923, C -138.909, E1 0.000, E2 0.0, E3 0.0, E4 0.0, E5 0.0, E6 0.0} C_DIS
>>>>>>>>>>>>>>>>>>>>>>>>>>>>GAS SUPPLY ON at=END
>>>>>>>>>>>>>>>>>>>>>>>>>>>>POWDER FEED ON at=END
>>>>>>>>>>>>>>>>>>>>>>>>>>>>LASER ON at=END
LIN {E6POS: X 1439.364, Y -12.200, Z 512.293, A 41.818, B 74.077, C -139.293, E1 0.000, E2 0.0, E3 0.0, E4 0.0, E5 0.0, E6 0.0} C_DIS
;POWDER FEED RATE  =  3.0
;LASER INTENSITY  =  4.0
LIN {E6POS: X 1430.258, Y -2.040, Z 512.293, A 41.966, B 73.600, C -139.215, E1 0.000, E2 0.0, E3 0.0, E4 0.0, E5 0.0, E6 0.0} C_DIS
;POWDER FEED RATE  =  3.0
;LASER INTENSITY  =  4.0
LIN {E6POS: X 1421.058, Y 8.120, Z 512.293, A 42.404, B 73.100, C -138.853, E1 0.000, E2 0.0, E3 0.0, E4 0.0, E5 0.0, E6 0.0} C_DIS
;POWDER FEED RATE  =  3.0
;LASER INTENSITY  =  4.0
LIN {E6POS: X 1411.670, Y 18.280, Z 512.293, A 43.120, B 72.662, C -138.207, E1 0.000, E2 0.0, E3 0.0, E4 0.0, E5 0.0, E6 0.0} C_DIS
;POWDER FEED RATE  =  3.0
;LASER INTENSITY  =  4.0
LIN {E6POS: X 1402.251, Y 28.440, Z 512.558, A 51.092, B 70.130, C -130.637, E1 0.000, E2 0.0, E3 0.0, E4 0.0, E5 0.0, E6 0.0} C_DIS
;POWDER FEED RATE  =  3.0
;LASER INTENSITY  =  4.0
LIN {E6POS: X 1393.968, Y 38.600, Z 514.412, A 65.218, B 62.820, C -117.429, E1 0.000, E2 0.0, E3 0.0, E4 0.0, E5 0.0, E6 0.0} C_DIS
;POWDER FEED RATE  =  3.0
;LASER INTENSITY  =  4.0
LIN {E6POS: X 1388.243, Y 48.760, Z 519.444, A 76.433, B 51.357, C -107.169, E1 0.000, E2 0.0, E3 0.0, E4 0.0, E5 0.0, E6 0.0} C_DIS
;POWDER FEED RATE  =  3.0
;LASER INTENSITY  =  4.0
LIN {E6POS: X 1385.831, Y 58.920, Z 528.449, A 81.926, B 43.726, C -101.598, E1 0.000, E2 0.0, E3 0.0, E4 0.0, E5 0.0, E6 0.0} C_DIS
;POWDER FEED RATE  =  3.0
;LASER INTENSITY  =  4.0
LIN {E6POS: X 1384.839, Y 69.080, Z 539.043, A 83.995, B 44.030, C -98.606, E1 0.000, E2 0.0, E3 0.0, E4 0.0, E5 0.0, E6 0.0} C_DIS
;POWDER FEED RATE  =  3.0
;LASER INTENSITY  =  4.0
LIN {E6POS: X 1382.710, Y 79.240, Z 548.048, A 83.677, B 53.622, C -97.836, E1 0.000, E2 0.0, E3 0.0, E4 0.0, E5 0.0, E6 0.0} C_DIS
;POWDER FEED RATE  =  3.0
;LASER INTENSITY  =  4.0
LIN {E6POS: X 1377.519, Y 89.400, Z 553.081, A 79.194, B 70.011, C -101.481, E1 0.000, E2 0.0, E3 0.0, E4 0.0, E5 0.0, E6 0.0} C_DIS
;POWDER FEED RATE  =  3.0
;LASER INTENSITY  =  4.0
LIN {E6POS: X 1369.866, Y 99.560, Z 554.935, A 63.965, B 81.644, C -116.277, E1 0.000, E2 0.0, E3 0.0, E4 0.0, E5 0.0, E6 0.0} C_DIS
;POWDER FEED RATE  =  3.0
;LASER INTENSITY  =  4.0
LIN {E6POS: X 1360.981, Y 109.720, Z 555.199, A 41.818, B 85.006, C -138.290, E1 0.000, E2 0.0, E3 0.0, E4 0.0, E5 0.0, E6 0.0} C_DIS
;POWDER FEED RATE  =  3.0
;LASER INTENSITY  =  4.0
LIN {E6POS: X 1351.891, Y 119.880, Z 555.199, A 41.818, B 84.895, C -138.295, E1 0.000, E2 0.0, E3 0.0, E4 0.0, E5 0.0, E6 0.0} C_DIS
;POWDER FEED RATE  =  3.0
;LASER INTENSITY  =  4.0
LIN {E6POS: X 1342.801, Y 130.040, Z 555.199, A 41.818, B 84.780, C -138.300, E1 0.000, E2 0.0, E3 0.0, E4 0.0, E5 0.0, E6 0.0} C_DIS
;POWDER FEED RATE  =  3.0
;LASER INTENSITY  =  4.0
LIN {E6POS: X 1333.711, Y 140.200, Z 555.199, A 41.818, B 84.659, C -138.306, E1 0.000, E2 0.0, E3 0.0, E4 0.0, E5 0.0, E6 0.0} C_DIS
;POWDER FEED RATE  =  3.0
;LASER INTENSITY  =  4.0
>>>>>>>>>>>>>>>>>>>>>>>>>>>>POWDER FEED OFF  at=START
>>>>>>>>>>>>>>>>>>>>>>>>>>>>LASER OFF at=START
>>>>>>>>>>>>>>>>>>>>>>>>>>>>GAS SUPPLY OFF  at=START
LIN {E6POS: X 1333.711, Y 140.200, Z 555.199, A 41.818, B 84.659, C -138.306, E1 0.000, E2 0.0, E3 0.0, E4 0.0, E5 0.0, E6 0.0} C_DIS
LIN {E6POS: X 1342.801, Y 130.040, Z 555.199, A 41.818, B 84.780, C -138.300, E1 0.000, E2 0.0, E3 0.0, E4 0.0, E5 0.0, E6 0.0} C_DIS
LIN {E6POS: X 1342.801, Y 130.040, Z 555.199, A 41.818, B 84.780, C -138.300, E1 0.000, E2 0.0, E3 0.0, E4 0.0, E5 0.0, E6 0.0} C_DIS
>>>>>>>>>>>>>>>>>>>>>>>>>>>>GAS SUPPLY ON at=END
>>>>>>>>>>>>>>>>>>>>>>>>>>>>POWDER FEED ON at=END
>>>>>>>>>>>>>>>>>>>>>>>>>>>>LASER ON at=END
LIN {E6POS: X 1444.830, Y -12.200, Z 513.531, A 42.284, B 72.073, C -139.132, E1 0.000, E2 0.0, E3 0.0, E4 0.0, E5 0.0, E6 0.0} C_DIS
;POWDER FEED RATE  =  3.0
;LASER INTENSITY  =  4.0
LIN {E6POS: X 1435.579, Y -2.040, Z 513.531, A 42.393, B 71.617, C -139.097, E1 0.000, E2 0.0, E3 0.0, E4 0.0, E5 0.0, E6 0.0} C_DIS
;POWDER FEED RATE  =  3.0
;LASER INTENSITY  =  4.0
LIN {E6POS: X 1426.256, Y 8.120, Z 513.531, A 42.718, B 71.153, C -138.852, E1 0.000, E2 0.0, E3 0.0, E4 0.0, E5 0.0, E6 0.0} C_DIS
;POWDER FEED RATE  =  3.0
;LASER INTENSITY  =  4.0
LIN {E6POS: X 1416.792, Y 18.280, Z 513.531, A 43.252, B 70.759, C -138.387, E1 0.000, E2 0.0, E3 0.0, E4 0.0, E5 0.0, E6 0.0} C_DIS
;POWDER FEED RATE  =  3.0
;LASER INTENSITY  =  4.0
LIN {E6POS: X 1407.376, Y 28.440, Z 513.791, A 50.003, B 68.519, C -132.039, E1 0.000, E2 0.0, E3 0.0, E4 0.0, E5 0.0, E6 0.0} C_DIS
;POWDER FEED RATE  =  3.0
;LASER INTENSITY  =  4.0
LIN {E6POS: X 1399.238, Y 38.600, Z 515.610, A 63.152, B 62.140, C -119.793, E1 0.000, E2 0.0, E3 0.0, E4 0.0, E5 0.0, E6 0.0} C_DIS
;POWDER FEED RATE  =  3.0
;LASER INTENSITY  =  4.0
LIN {E6POS: X 1393.867, Y 48.760, Z 520.550, A 74.931, B 51.747, C -108.924, E1 0.000, E2 0.0, E3 0.0, E4 0.0, E5 0.0, E6 0.0} C_DIS
;POWDER FEED RATE  =  3.0
;LASER INTENSITY  =  4.0
LIN {E6POS: X 1392.044, Y 58.920, Z 529.389, A 81.237, B 44.453, C -102.413, E1 0.000, E2 0.0, E3 0.0, E4 0.0, E5 0.0, E6 0.0} C_DIS
;POWDER FEED RATE  =  3.0
;LASER INTENSITY  =  4.0
LIN {E6POS: X 1391.711, Y 69.080, Z 539.789, A 83.836, B 44.737, C -98.723, E1 0.000, E2 0.0, E3 0.0, E4 0.0, E5 0.0, E6 0.0} C_DIS
;POWDER FEED RATE  =  3.0
;LASER INTENSITY  =  4.0
LIN {E6POS: X 1390.101, Y 79.240, Z 548.628, A 83.964, B 54.304, C -97.418, E1 0.000, E2 0.0, E3 0.0, E4 0.0, E5 0.0, E6 0.0} C_DIS
;POWDER FEED RATE  =  3.0
;LASER INTENSITY  =  4.0
LIN {E6POS: X 1385.132, Y 89.400, Z 553.567, A 80.200, B 70.679, C -100.373, E1 0.000, E2 0.0, E3 0.0, E4 0.0, E5 0.0, E6 0.0} C_DIS
;POWDER FEED RATE  =  3.0
;LASER INTENSITY  =  4.0
LIN {E6POS: X 1377.465, Y 99.560, Z 555.387, A 66.005, B 82.340, C -114.186, E1 0.000, E2 0.0, E3 0.0, E4 0.0, E5 0.0, E6 0.0} C_DIS
;POWDER FEED RATE  =  3.0
;LASER INTENSITY  =  4.0
LIN {E6POS: X 1368.451, Y 109.720, Z 555.647, A 42.284, B 85.761, C -137.794, E1 0.000, E2 0.0, E3 0.0, E4 0.0, E5 0.0, E6 0.0} C_DIS
;POWDER FEED RATE  =  3.0
;LASER INTENSITY  =  4.0
LIN {E6POS: X 1359.211, Y 119.880, Z 555.647, A 42.284, B 85.683, C -137.797, E1 0.000, E2 0.0, E3 0.0, E4 0.0, E5 0.0, E6 0.0} C_DIS
;POWDER FEED RATE  =  3.0
;LASER INTENSITY  =  4.0
LIN {E6POS: X 1349.971, Y 130.040, Z 555.647, A 42.284, B 85.601, C -137.800, E1 0.000, E2 0.0, E3 0.0, E4 0.0, E5 0.0, E6 0.0} C_DIS
;POWDER FEED RATE  =  3.0
;LASER INTENSITY  =  4.0
LIN {E6POS: X 1340.732, Y 140.200, Z 555.647, A 42.284, B 85.516, C -137.804, E1 0.000, E2 0.0, E3 0.0, E4 0.0, E5 0.0, E6 0.0} C_DIS
;POWDER FEED RATE  =  3.0
;LASER INTENSITY  =  4.0
>>>>>>>>>>>>>>>>>>>>>>>>>>>>POWDER FEED OFF  at=START
>>>>>>>>>>>>>>>>>>>>>>>>>>>>LASER OFF at=START
>>>>>>>>>>>>>>>>>>>>>>>>>>>>GAS SUPPLY OFF  at=START
LIN {E6POS: X 1340.732, Y 140.200, Z 555.647, A 42.284, B 85.516, C -137.804, E1 0.000, E2 0.0, E3 0.0, E4 0.0, E5 0.0, E6 0.0} C_DIS
LIN {E6POS: X 1349.971, Y 130.040, Z 555.647, A 42.284, B 85.601, C -137.800, E1 0.000, E2 0.0, E3 0.0, E4 0.0, E5 0.0, E6 0.0} C_DIS
LIN {E6POS: X 1349.971, Y 130.040, Z 555.647, A 42.284, B 85.601, C -137.800, E1 0.000, E2 0.0, E3 0.0, E4 0.0, E5 0.0, E6 0.0} C_DIS
>>>>>>>>>>>>>>>>>>>>>>>>>>>>GAS SUPPLY ON at=END
>>>>>>>>>>>>>>>>>>>>>>>>>>>>POWDER FEED ON at=END
>>>>>>>>>>>>>>>>>>>>>>>>>>>>LASER ON at=END
LIN {E6POS: X 1450.032, Y -12.200, Z 514.827, A 42.660, B 70.687, C -138.989, E1 0.000, E2 0.0, E3 0.0, E4 0.0, E5 0.0, E6 0.0} C_DIS
;POWDER FEED RATE  =  3.0
;LASER INTENSITY  =  4.0
LIN {E6POS: X 1440.661, Y -2.040, Z 514.827, A 42.738, B 70.282, C -138.982, E1 0.000, E2 0.0, E3 0.0, E4 0.0, E5 0.0, E6 0.0} C_DIS
;POWDER FEED RATE  =  3.0
;LASER INTENSITY  =  4.0
LIN {E6POS: X 1431.239, Y 8.120, Z 514.827, A 42.973, B 69.879, C -138.822, E1 0.000, E2 0.0, E3 0.0, E4 0.0, E5 0.0, E6 0.0} C_DIS
;POWDER FEED RATE  =  3.0
;LASER INTENSITY  =  4.0
LIN {E6POS: X 1421.713, Y 18.280, Z 514.827, A 43.360, B 69.549, C -138.497, E1 0.000, E2 0.0, E3 0.0, E4 0.0, E5 0.0, E6 0.0} C_DIS
;POWDER FEED RATE  =  3.0
;LASER INTENSITY  =  4.0
LIN {E6POS: X 1412.303, Y 28.440, Z 515.082, A 49.262, B 67.560, C -132.980, E1 0.000, E2 0.0, E3 0.0, E4 0.0, E5 0.0, E6 0.0} C_DIS
;POWDER FEED RATE  =  3.0
;LASER INTENSITY  =  4.0
LIN {E6POS: X 1404.303, Y 38.600, Z 516.861, A 61.613, B 61.920, C -121.488, E1 0.000, E2 0.0, E3 0.0, E4 0.0, E5 0.0, E6 0.0} C_DIS
;POWDER FEED RATE  =  3.0
;LASER INTENSITY  =  4.0
LIN {E6POS: X 1399.280, Y 48.760, Z 521.692, A 73.745, B 52.391, C -110.206, E1 0.000, E2 0.0, E3 0.0, E4 0.0, E5 0.0, E6 0.0} C_DIS
;POWDER FEED RATE  =  3.0
;LASER INTENSITY  =  4.0
LIN {E6POS: X 1398.044, Y 58.920, Z 530.336, A 80.713, B 45.340, C -102.947, E1 0.000, E2 0.0, E3 0.0, E4 0.0, E5 0.0, E6 0.0} C_DIS
;POWDER FEED RATE  =  3.0
;LASER INTENSITY  =  4.0
LIN {E6POS: X 1398.374, Y 69.080, Z 540.505, A 83.766, B 45.566, C -98.698, E1 0.000, E2 0.0, E3 0.0, E4 0.0, E5 0.0, E6 0.0} C_DIS
;POWDER FEED RATE  =  3.0
;LASER INTENSITY  =  4.0
LIN {E6POS: X 1397.292, Y 79.240, Z 549.149, A 84.293, B 55.082, C -96.948, E1 0.000, E2 0.0, E3 0.0, E4 0.0, E5 0.0, E6 0.0} C_DIS
;POWDER FEED RATE  =  3.0
;LASER INTENSITY  =  4.0
LIN {E6POS: X 1392.562, Y 89.400, Z 553.980, A 81.226, B 71.388, C -99.250, E1 0.000, E2 0.0, E3 0.0, E4 0.0, E5 0.0, E6 0.0} C_DIS
;POWDER FEED RATE  =  3.0
;LASER INTENSITY  =  4.0
LIN {E6POS: X 1384.907, Y 99.560, Z 555.760, A 68.210, B 83.021, C -111.937, E1 0.000, E2 0.0, E3 0.0, E4 0.0, E5 0.0, E6 0.0} C_DIS
;POWDER FEED RATE  =  3.0
;LASER INTENSITY  =  4.0
LIN {E6POS: X 1375.788, Y 109.720, Z 556.014, A 42.660, B 86.485, C -137.394, E1 0.000, E2 0.0, E3 0.0, E4 0.0, E5 0.0, E6 0.0} C_DIS
;POWDER FEED RATE  =  3.0
;LASER INTENSITY  =  4.0
LIN {E6POS: X 1366.426, Y 119.880, Z 556.014, A 42.660, B 86.431, C -137.396, E1 0.000, E2 0.0, E3 0.0, E4 0.0, E5 0.0, E6 0.0} C_DIS
;POWDER FEED RATE  =  3.0
;LASER INTENSITY  =  4.0
LIN {E6POS: X 1357.064, Y 130.040, Z 556.014, A 42.660, B 86.375, C -137.398, E1 0.000, E2 0.0, E3 0.0, E4 0.0, E5 0.0, E6 0.0} C_DIS
;POWDER FEED RATE  =  3.0
;LASER INTENSITY  =  4.0
LIN {E6POS: X 1347.702, Y 140.200, Z 556.014, A 42.660, B 86.318, C -137.399, E1 0.000, E2 0.0, E3 0.0, E4 0.0, E5 0.0, E6 0.0} C_DIS
;POWDER FEED RATE  =  3.0
;LASER INTENSITY  =  4.0
>>>>>>>>>>>>>>>>>>>>>>>>>>>>POWDER FEED OFF  at=START
>>>>>>>>>>>>>>>>>>>>>>>>>>>>LASER OFF at=START
>>>>>>>>>>>>>>>>>>>>>>>>>>>>GAS SUPPLY OFF  at=START
LIN {E6POS: X 1347.702, Y 140.200, Z 556.014, A 42.660, B 86.318, C -137.399, E1 0.000, E2 0.0, E3 0.0, E4 0.0, E5 0.0, E6 0.0} C_DIS
LIN {E6POS: X 1357.064, Y 130.040, Z 556.014, A 42.660, B 86.375, C -137.398, E1 0.000, E2 0.0, E3 0.0, E4 0.0, E5 0.0, E6 0.0} C_DIS
LIN {E6POS: X 1357.064, Y 130.040, Z 556.014, A 42.660, B 86.375, C -137.398, E1 0.000, E2 0.0, E3 0.0, E4 0.0, E5 0.0, E6 0.0} C_DIS
>>>>>>>>>>>>>>>>>>>>>>>>>>>>GAS SUPPLY ON at=END
>>>>>>>>>>>>>>>>>>>>>>>>>>>>POWDER FEED ON at=END
>>>>>>>>>>>>>>>>>>>>>>>>>>>>LASER ON at=END
